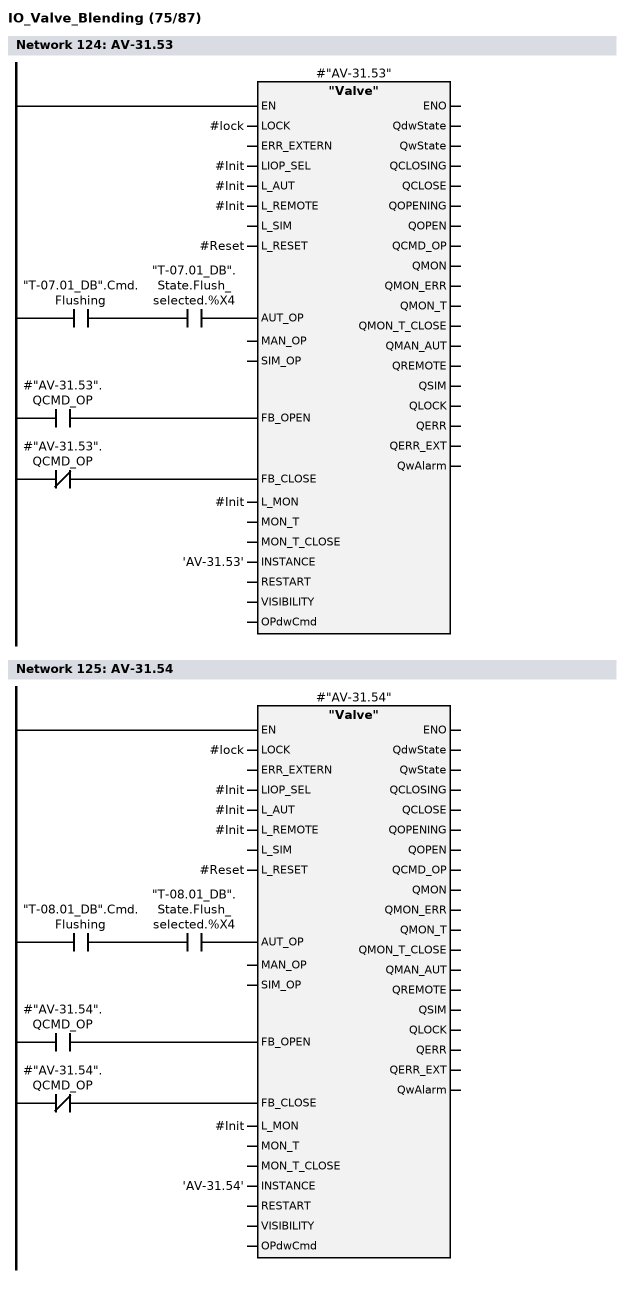
   RUNG wire#powerrail
      #"AV-31.53"(AUT_OP := wire#w1, FB_OPEN := wire#w2, FB_CLOSE := wire#w3, LOCK := #lock, ERR_EXTERN :=, LIOP_SEL := #Init, L_AUT := #Init, L_REMOTE := #Init, L_SIM :=, L_RESET := #Reset, MAN_OP :=, SIM_OP :=, L_MON := #Init, MON_T :=, MON_T_CLOSE :=, INSTANCE := 'AV-31.53', RESTART :=, VISIBILITY :=, OPdwCmd :=, QdwState =>, QwState =>, QCLOSING =>, QCLOSE =>, QOPENING =>, QOPEN =>, QCMD_OP =>, QMON =>, QMON_ERR =>, QMON_T =>, QMON_T_CLOSE =>, QMAN_AUT =>, QREMOTE =>, QSIM =>, QLOCK =>, QERR =>, QERR_EXT =>, QwAlarm =>)
   END_RUNG
   RUNG wire#powerrail
      Contact( "T-07.01_DB".Cmd.Flushing )
      Contact( "T-07.01_DB".State.Flush_selected.%X4 )
   END_RUNG wire#w1
   RUNG wire#powerrail
      Contact( #"AV-31.53".QCMD_OP )
   END_RUNG wire#w2
   RUNG wire#powerrail
      I_Contact( #"AV-31.53".QCMD_OP )
   END_RUNG wire#w3
   // the same network as SCL:
   #"AV-31.53"(LOCK := #lock,   // "Valve"
               LIOP_SEL := #Init,
               L_AUT := #Init,
               L_REMOTE := #Init,
               L_RESET := #Reset,
               AUT_OP := "T-07.01_DB".Cmd.Flushing AND "T-07.01_DB".State.Flush_selected.%X4,
               FB_OPEN := #"AV-31.53".QCMD_OP,
               FB_CLOSE := NOT #"AV-31.53".QCMD_OP,
               L_MON := #Init,
               INSTANCE := 'AV-31.53');
END_REGION

REGION Network 125: AV-31.54
   RUNG wire#powerrail
      #"AV-31.54"(AUT_OP := wire#w1, FB_OPEN := wire#w2, FB_CLOSE := wire#w3, LOCK := #lock, ERR_EXTERN :=, LIOP_SEL := #Init, L_AUT := #Init, L_REMOTE := #Init, L_SIM :=, L_RESET := #Reset, MAN_OP :=, SIM_OP :=, L_MON := #Init, MON_T :=, MON_T_CLOSE :=, INSTANCE := 'AV-31.54', RESTART :=, VISIBILITY :=, OPdwCmd :=, QdwState =>, QwState =>, QCLOSING =>, QCLOSE =>, QOPENING =>, QOPEN =>, QCMD_OP =>, QMON =>, QMON_ERR =>, QMON_T =>, QMON_T_CLOSE =>, QMAN_AUT =>, QREMOTE =>, QSIM =>, QLOCK =>, QERR =>, QERR_EXT =>, QwAlarm =>)
   END_RUNG
   RUNG wire#powerrail
      Contact( "T-08.01_DB".Cmd.Flushing )
      Contact( "T-08.01_DB".State.Flush_selected.%X4 )
   END_RUNG wire#w1
   RUNG wire#powerrail
      Contact( #"AV-31.54".QCMD_OP )
   END_RUNG wire#w2
   RUNG wire#powerrail
      I_Contact( #"AV-31.54".QCMD_OP )
   END_RUNG wire#w3
   // the same network as SCL:
   #"AV-31.54"(LOCK := #lock,   // "Valve"
               LIOP_SEL := #Init,
               L_AUT := #Init,
               L_REMOTE := #Init,
               L_RESET := #Reset,
               AUT_OP := "T-08.01_DB".Cmd.Flushing AND "T-08.01_DB".State.Flush_selected.%X4,
               FB_OPEN := #"AV-31.54".QCMD_OP,
               FB_CLOSE := NOT #"AV-31.54".QCMD_OP,
               L_MON := #Init,
               INSTANCE := 'AV-31.54');
END_REGION

REGION Network 126: AV-31.55
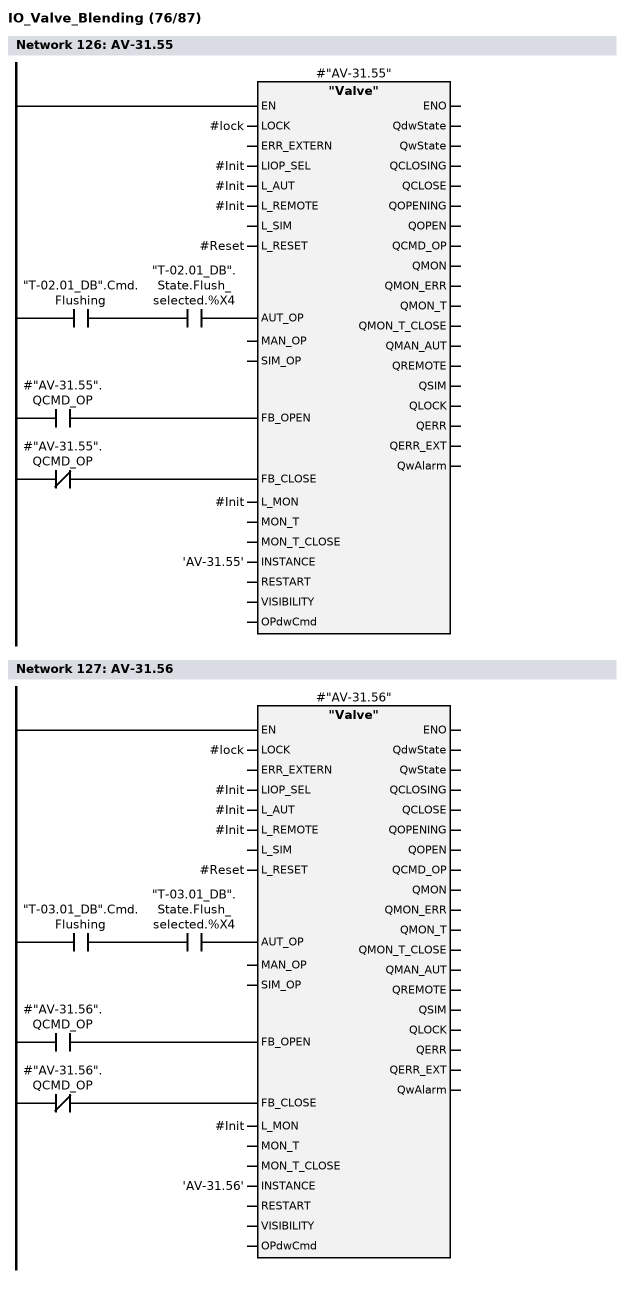
   RUNG wire#powerrail
      #"AV-31.55"(AUT_OP := wire#w1, FB_OPEN := wire#w2, FB_CLOSE := wire#w3, LOCK := #lock, ERR_EXTERN :=, LIOP_SEL := #Init, L_AUT := #Init, L_REMOTE := #Init, L_SIM :=, L_RESET := #Reset, MAN_OP :=, SIM_OP :=, L_MON := #Init, MON_T :=, MON_T_CLOSE :=, INSTANCE := 'AV-31.55', RESTART :=, VISIBILITY :=, OPdwCmd :=, QdwState =>, QwState =>, QCLOSING =>, QCLOSE =>, QOPENING =>, QOPEN =>, QCMD_OP =>, QMON =>, QMON_ERR =>, QMON_T =>, QMON_T_CLOSE =>, QMAN_AUT =>, QREMOTE =>, QSIM =>, QLOCK =>, QERR =>, QERR_EXT =>, QwAlarm =>)
   END_RUNG
   RUNG wire#powerrail
      Contact( "T-02.01_DB".Cmd.Flushing )
      Contact( "T-02.01_DB".State.Flush_selected.%X4 )
   END_RUNG wire#w1
   RUNG wire#powerrail
      Contact( #"AV-31.55".QCMD_OP )
   END_RUNG wire#w2
   RUNG wire#powerrail
      I_Contact( #"AV-31.55".QCMD_OP )
   END_RUNG wire#w3
   // the same network as SCL:
   #"AV-31.55"(LOCK := #lock,   // "Valve"
               LIOP_SEL := #Init,
               L_AUT := #Init,
               L_REMOTE := #Init,
               L_RESET := #Reset,
               AUT_OP := "T-02.01_DB".Cmd.Flushing AND "T-02.01_DB".State.Flush_selected.%X4,
               FB_OPEN := #"AV-31.55".QCMD_OP,
               FB_CLOSE := NOT #"AV-31.55".QCMD_OP,
               L_MON := #Init,
               INSTANCE := 'AV-31.55');
END_REGION

REGION Network 127: AV-31.56
   RUNG wire#powerrail
      #"AV-31.56"(AUT_OP := wire#w1, FB_OPEN := wire#w2, FB_CLOSE := wire#w3, LOCK := #lock, ERR_EXTERN :=, LIOP_SEL := #Init, L_AUT := #Init, L_REMOTE := #Init, L_SIM :=, L_RESET := #Reset, MAN_OP :=, SIM_OP :=, L_MON := #Init, MON_T :=, MON_T_CLOSE :=, INSTANCE := 'AV-31.56', RESTART :=, VISIBILITY :=, OPdwCmd :=, QdwState =>, QwState =>, QCLOSING =>, QCLOSE =>, QOPENING =>, QOPEN =>, QCMD_OP =>, QMON =>, QMON_ERR =>, QMON_T =>, QMON_T_CLOSE =>, QMAN_AUT =>, QREMOTE =>, QSIM =>, QLOCK =>, QERR =>, QERR_EXT =>, QwAlarm =>)
   END_RUNG
   RUNG wire#powerrail
      Contact( "T-03.01_DB".Cmd.Flushing )
      Contact( "T-03.01_DB".State.Flush_selected.%X4 )
   END_RUNG wire#w1
   RUNG wire#powerrail
      Contact( #"AV-31.56".QCMD_OP )
   END_RUNG wire#w2
   RUNG wire#powerrail
      I_Contact( #"AV-31.56".QCMD_OP )
   END_RUNG wire#w3
   // the same network as SCL:
   #"AV-31.56"(LOCK := #lock,   // "Valve"
               LIOP_SEL := #Init,
               L_AUT := #Init,
               L_REMOTE := #Init,
               L_RESET := #Reset,
               AUT_OP := "T-03.01_DB".Cmd.Flushing AND "T-03.01_DB".State.Flush_selected.%X4,
               FB_OPEN := #"AV-31.56".QCMD_OP,
               FB_CLOSE := NOT #"AV-31.56".QCMD_OP,
               L_MON := #Init,
               INSTANCE := 'AV-31.56');
END_REGION

REGION Network 128: AV-31.57
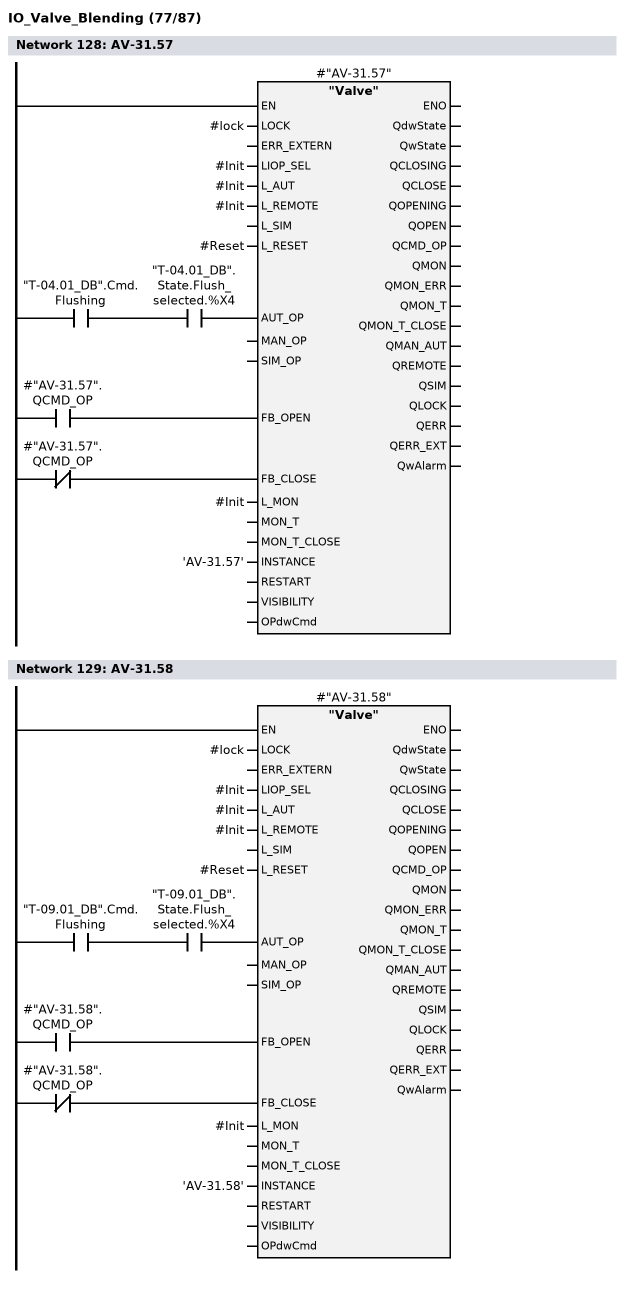
   RUNG wire#powerrail
      #"AV-31.57"(AUT_OP := wire#w1, FB_OPEN := wire#w2, FB_CLOSE := wire#w3, LOCK := #lock, ERR_EXTERN :=, LIOP_SEL := #Init, L_AUT := #Init, L_REMOTE := #Init, L_SIM :=, L_RESET := #Reset, MAN_OP :=, SIM_OP :=, L_MON := #Init, MON_T :=, MON_T_CLOSE :=, INSTANCE := 'AV-31.57', RESTART :=, VISIBILITY :=, OPdwCmd :=, QdwState =>, QwState =>, QCLOSING =>, QCLOSE =>, QOPENING =>, QOPEN =>, QCMD_OP =>, QMON =>, QMON_ERR =>, QMON_T =>, QMON_T_CLOSE =>, QMAN_AUT =>, QREMOTE =>, QSIM =>, QLOCK =>, QERR =>, QERR_EXT =>, QwAlarm =>)
   END_RUNG
   RUNG wire#powerrail
      Contact( "T-04.01_DB".Cmd.Flushing )
      Contact( "T-04.01_DB".State.Flush_selected.%X4 )
   END_RUNG wire#w1
   RUNG wire#powerrail
      Contact( #"AV-31.57".QCMD_OP )
   END_RUNG wire#w2
   RUNG wire#powerrail
      I_Contact( #"AV-31.57".QCMD_OP )
   END_RUNG wire#w3
   // the same network as SCL:
   #"AV-31.57"(LOCK := #lock,   // "Valve"
               LIOP_SEL := #Init,
               L_AUT := #Init,
               L_REMOTE := #Init,
               L_RESET := #Reset,
               AUT_OP := "T-04.01_DB".Cmd.Flushing AND "T-04.01_DB".State.Flush_selected.%X4,
               FB_OPEN := #"AV-31.57".QCMD_OP,
               FB_CLOSE := NOT #"AV-31.57".QCMD_OP,
               L_MON := #Init,
               INSTANCE := 'AV-31.57');
END_REGION

REGION Network 129: AV-31.58
   RUNG wire#powerrail
      #"AV-31.58"(AUT_OP := wire#w1, FB_OPEN := wire#w2, FB_CLOSE := wire#w3, LOCK := #lock, ERR_EXTERN :=, LIOP_SEL := #Init, L_AUT := #Init, L_REMOTE := #Init, L_SIM :=, L_RESET := #Reset, MAN_OP :=, SIM_OP :=, L_MON := #Init, MON_T :=, MON_T_CLOSE :=, INSTANCE := 'AV-31.58', RESTART :=, VISIBILITY :=, OPdwCmd :=, QdwState =>, QwState =>, QCLOSING =>, QCLOSE =>, QOPENING =>, QOPEN =>, QCMD_OP =>, QMON =>, QMON_ERR =>, QMON_T =>, QMON_T_CLOSE =>, QMAN_AUT =>, QREMOTE =>, QSIM =>, QLOCK =>, QERR =>, QERR_EXT =>, QwAlarm =>)
   END_RUNG
   RUNG wire#powerrail
      Contact( "T-09.01_DB".Cmd.Flushing )
      Contact( "T-09.01_DB".State.Flush_selected.%X4 )
   END_RUNG wire#w1
   RUNG wire#powerrail
      Contact( #"AV-31.58".QCMD_OP )
   END_RUNG wire#w2
   RUNG wire#powerrail
      I_Contact( #"AV-31.58".QCMD_OP )
   END_RUNG wire#w3
   // the same network as SCL:
   #"AV-31.58"(LOCK := #lock,   // "Valve"
               LIOP_SEL := #Init,
               L_AUT := #Init,
               L_REMOTE := #Init,
               L_RESET := #Reset,
               AUT_OP := "T-09.01_DB".Cmd.Flushing AND "T-09.01_DB".State.Flush_selected.%X4,
               FB_OPEN := #"AV-31.58".QCMD_OP,
               FB_CLOSE := NOT #"AV-31.58".QCMD_OP,
               L_MON := #Init,
               INSTANCE := 'AV-31.58');
END_REGION

REGION Network 130: AV-31.59
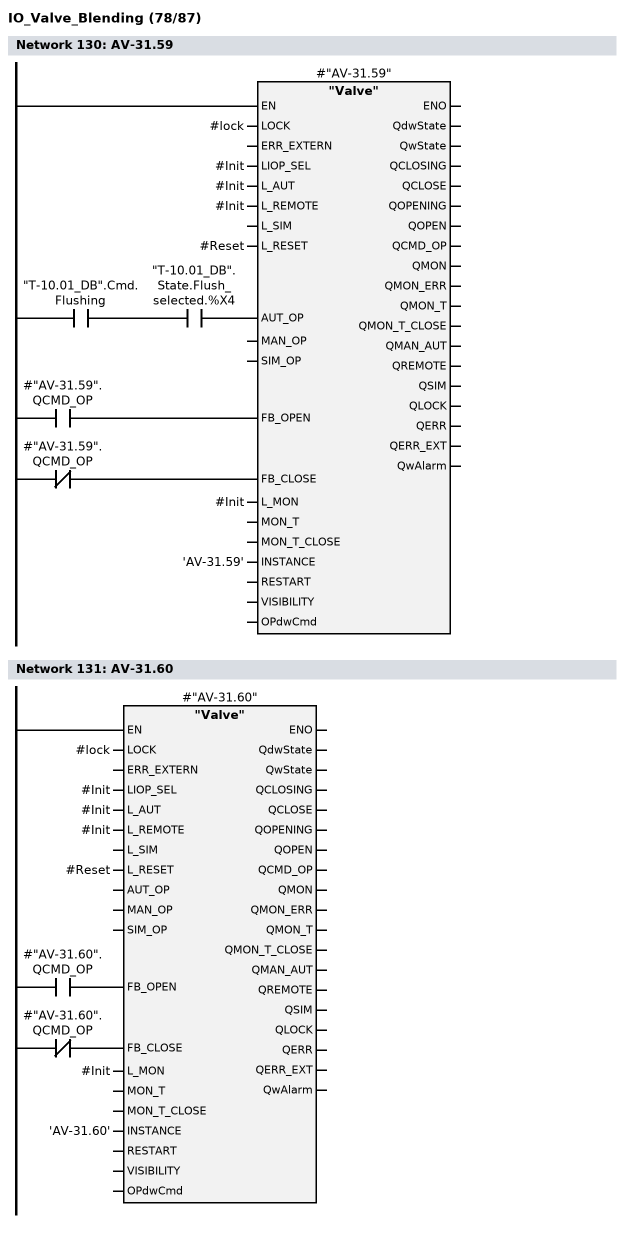
   RUNG wire#powerrail
      #"AV-31.59"(AUT_OP := wire#w1, FB_OPEN := wire#w2, FB_CLOSE := wire#w3, LOCK := #lock, ERR_EXTERN :=, LIOP_SEL := #Init, L_AUT := #Init, L_REMOTE := #Init, L_SIM :=, L_RESET := #Reset, MAN_OP :=, SIM_OP :=, L_MON := #Init, MON_T :=, MON_T_CLOSE :=, INSTANCE := 'AV-31.59', RESTART :=, VISIBILITY :=, OPdwCmd :=, QdwState =>, QwState =>, QCLOSING =>, QCLOSE =>, QOPENING =>, QOPEN =>, QCMD_OP =>, QMON =>, QMON_ERR =>, QMON_T =>, QMON_T_CLOSE =>, QMAN_AUT =>, QREMOTE =>, QSIM =>, QLOCK =>, QERR =>, QERR_EXT =>, QwAlarm =>)
   END_RUNG
   RUNG wire#powerrail
      Contact( "T-10.01_DB".Cmd.Flushing )
      Contact( "T-10.01_DB".State.Flush_selected.%X4 )
   END_RUNG wire#w1
   RUNG wire#powerrail
      Contact( #"AV-31.59".QCMD_OP )
   END_RUNG wire#w2
   RUNG wire#powerrail
      I_Contact( #"AV-31.59".QCMD_OP )
   END_RUNG wire#w3
   // the same network as SCL:
   #"AV-31.59"(LOCK := #lock,   // "Valve"
               LIOP_SEL := #Init,
               L_AUT := #Init,
               L_REMOTE := #Init,
               L_RESET := #Reset,
               AUT_OP := "T-10.01_DB".Cmd.Flushing AND "T-10.01_DB".State.Flush_selected.%X4,
               FB_OPEN := #"AV-31.59".QCMD_OP,
               FB_CLOSE := NOT #"AV-31.59".QCMD_OP,
               L_MON := #Init,
               INSTANCE := 'AV-31.59');
END_REGION

REGION Network 131: AV-31.60
   RUNG wire#powerrail
      #"AV-31.60"(FB_OPEN := wire#w1, FB_CLOSE := wire#w2, LOCK := #lock, ERR_EXTERN :=, LIOP_SEL := #Init, L_AUT := #Init, L_REMOTE := #Init, L_SIM :=, L_RESET := #Reset, AUT_OP :=, MAN_OP :=, SIM_OP :=, L_MON := #Init, MON_T :=, MON_T_CLOSE :=, INSTANCE := 'AV-31.60', RESTART :=, VISIBILITY :=, OPdwCmd :=, QdwState =>, QwState =>, QCLOSING =>, QCLOSE =>, QOPENING =>, QOPEN =>, QCMD_OP =>, QMON =>, QMON_ERR =>, QMON_T =>, QMON_T_CLOSE =>, QMAN_AUT =>, QREMOTE =>, QSIM =>, QLOCK =>, QERR =>, QERR_EXT =>, QwAlarm =>)
   END_RUNG
   RUNG wire#powerrail
      Contact( #"AV-31.60".QCMD_OP )
   END_RUNG wire#w1
   RUNG wire#powerrail
      I_Contact( #"AV-31.60".QCMD_OP )
   END_RUNG wire#w2
   // the same network as SCL:
   #"AV-31.60"(LOCK := #lock,   // "Valve"
               LIOP_SEL := #Init,
               L_AUT := #Init,
               L_REMOTE := #Init,
               L_RESET := #Reset,
               FB_OPEN := #"AV-31.60".QCMD_OP,
               FB_CLOSE := NOT #"AV-31.60".QCMD_OP,
               L_MON := #Init,
               INSTANCE := 'AV-31.60');
END_REGION

REGION Network 132: AV-31.61
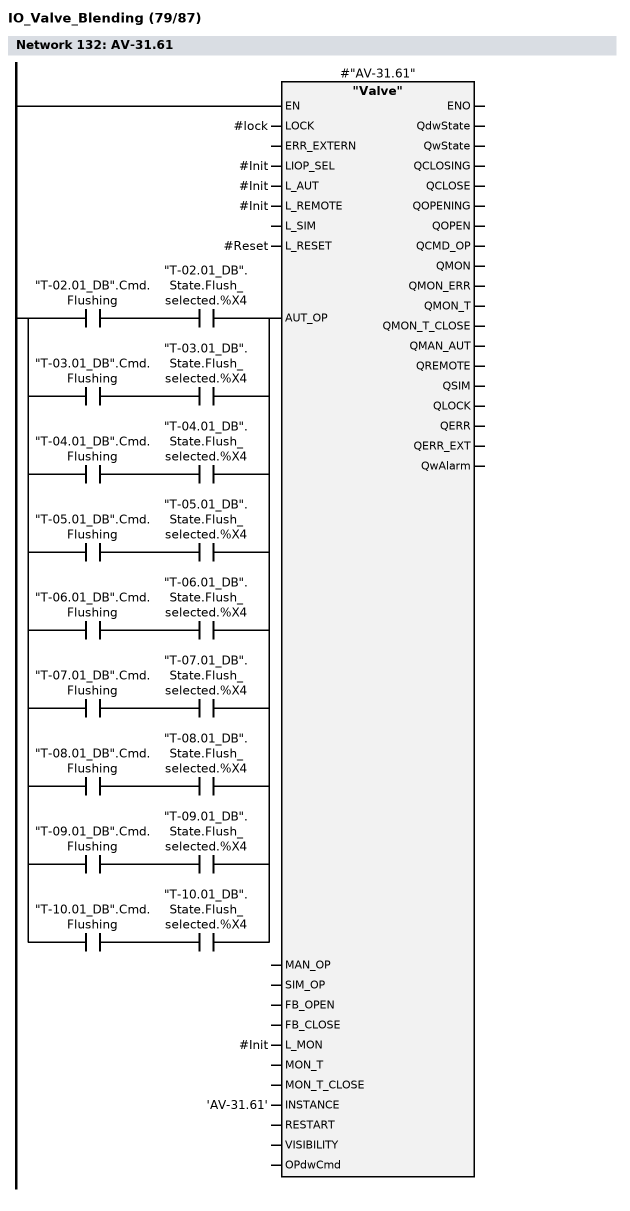
   RUNG wire#powerrail
      #"AV-31.61"(AUT_OP := wire#w1, LOCK := #lock, ERR_EXTERN :=, LIOP_SEL := #Init, L_AUT := #Init, L_REMOTE := #Init, L_SIM :=, L_RESET := #Reset, MAN_OP :=, SIM_OP :=, FB_OPEN :=, FB_CLOSE :=, L_MON := #Init, MON_T :=, MON_T_CLOSE :=, INSTANCE := 'AV-31.61', RESTART :=, VISIBILITY :=, OPdwCmd :=, QdwState =>, QwState =>, QCLOSING =>, QCLOSE =>, QOPENING =>, QOPEN =>, QCMD_OP =>, QMON =>, QMON_ERR =>, QMON_T =>, QMON_T_CLOSE =>, QMAN_AUT =>, QREMOTE =>, QSIM =>, QLOCK =>, QERR =>, QERR_EXT =>, QwAlarm =>)
   END_RUNG
   RUNG wire#powerrail
      Contact( "T-02.01_DB".Cmd.Flushing )
      Contact( "T-02.01_DB".State.Flush_selected.%X4 )
   END_RUNG wire#w1
   RUNG wire#powerrail
      Contact( "T-03.01_DB".Cmd.Flushing )
      Contact( "T-03.01_DB".State.Flush_selected.%X4 )
   END_RUNG wire#w1
   RUNG wire#powerrail
      Contact( "T-04.01_DB".Cmd.Flushing )
      Contact( "T-04.01_DB".State.Flush_selected.%X4 )
   END_RUNG wire#w1
   RUNG wire#powerrail
      Contact( "T-05.01_DB".Cmd.Flushing )
      Contact( "T-05.01_DB".State.Flush_selected.%X4 )
   END_RUNG wire#w1
   RUNG wire#powerrail
      Contact( "T-06.01_DB".Cmd.Flushing )
      Contact( "T-06.01_DB".State.Flush_selected.%X4 )
   END_RUNG wire#w1
   RUNG wire#powerrail
      Contact( "T-07.01_DB".Cmd.Flushing )
      Contact( "T-07.01_DB".State.Flush_selected.%X4 )
   END_RUNG wire#w1
   RUNG wire#powerrail
      Contact( "T-08.01_DB".Cmd.Flushing )
      Contact( "T-08.01_DB".State.Flush_selected.%X4 )
   END_RUNG wire#w1
   RUNG wire#powerrail
      Contact( "T-09.01_DB".Cmd.Flushing )
      Contact( "T-09.01_DB".State.Flush_selected.%X4 )
   END_RUNG wire#w1
   RUNG wire#powerrail
      Contact( "T-10.01_DB".Cmd.Flushing )
      Contact( "T-10.01_DB".State.Flush_selected.%X4 )
   END_RUNG wire#w1
   // the same network as SCL:
   #"AV-31.61"(LOCK := #lock,   // "Valve"
               LIOP_SEL := #Init,
               L_AUT := #Init,
               L_REMOTE := #Init,
               L_RESET := #Reset,
               AUT_OP := ("T-02.01_DB".Cmd.Flushing AND "T-02.01_DB".State.Flush_selected.%X4) OR ("T-03.01_DB".Cmd.Flushing AND "T-03.01_DB".State.Flush_selected.%X4) OR ("T-04.01_DB".Cmd.Flushing AND "T-04.01_DB".State.Flush_selected.%X4) OR ("T-05.01_DB".Cmd.Flushing AND "T-05.01_DB".State.Flush_selected.%X4) OR ("T-06.01_DB".Cmd.Flushing AND "T-06.01_DB".State.Flush_selected.%X4) OR ("T-07.01_DB".Cmd.Flushing AND "T-07.01_DB".State.Flush_selected.%X4) OR ("T-08.01_DB".Cmd.Flushing AND "T-08.01_DB".State.Flush_selected.%X4) OR ("T-09.01_DB".Cmd.Flushing AND "T-09.01_DB".State.Flush_selected.%X4) OR ("T-10.01_DB".Cmd.Flushing AND "T-10.01_DB".State.Flush_selected.%X4),
               L_MON := #Init,
               INSTANCE := 'AV-31.61');
END_REGION

REGION Network 133: AV-31.62
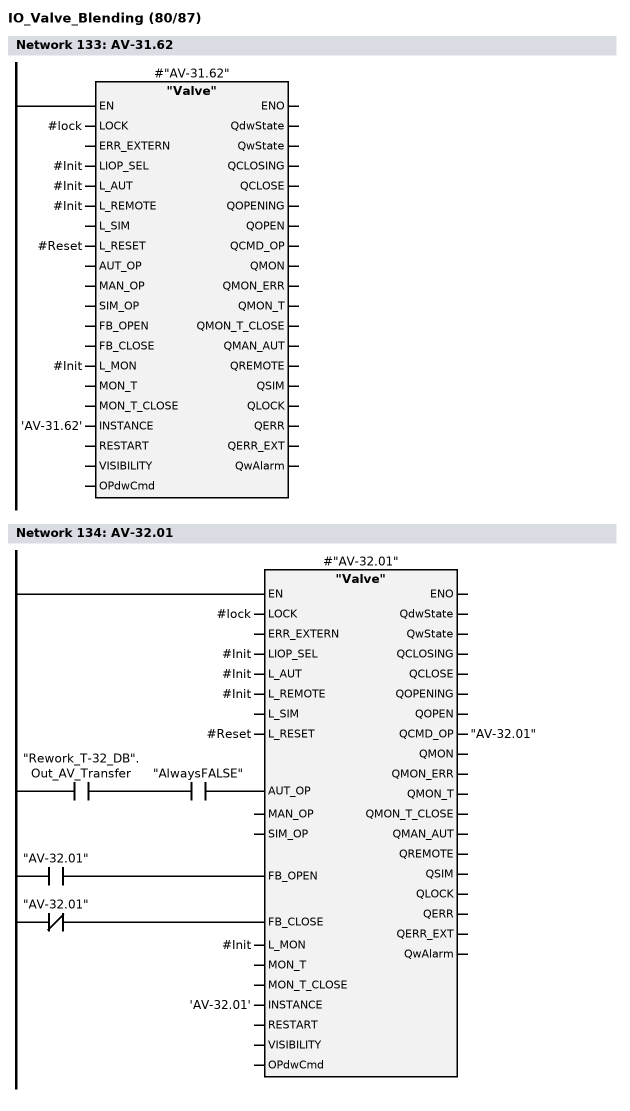
   RUNG wire#powerrail
      #"AV-31.62"(LOCK := #lock, ERR_EXTERN :=, LIOP_SEL := #Init, L_AUT := #Init, L_REMOTE := #Init, L_SIM :=, L_RESET := #Reset, AUT_OP :=, MAN_OP :=, SIM_OP :=, FB_OPEN :=, FB_CLOSE :=, L_MON := #Init, MON_T :=, MON_T_CLOSE :=, INSTANCE := 'AV-31.62', RESTART :=, VISIBILITY :=, OPdwCmd :=, QdwState =>, QwState =>, QCLOSING =>, QCLOSE =>, QOPENING =>, QOPEN =>, QCMD_OP =>, QMON =>, QMON_ERR =>, QMON_T =>, QMON_T_CLOSE =>, QMAN_AUT =>, QREMOTE =>, QSIM =>, QLOCK =>, QERR =>, QERR_EXT =>, QwAlarm =>)
   END_RUNG
   // the same network as SCL:
   #"AV-31.62"(LOCK := #lock,   // "Valve"
               LIOP_SEL := #Init,
               L_AUT := #Init,
               L_REMOTE := #Init,
               L_RESET := #Reset,
               L_MON := #Init,
               INSTANCE := 'AV-31.62');
END_REGION

REGION Network 134: AV-32.01
   RUNG wire#powerrail
      #"AV-32.01"(AUT_OP := wire#w1, FB_OPEN := wire#w2, FB_CLOSE := wire#w3, LOCK := #lock, ERR_EXTERN :=, LIOP_SEL := #Init, L_AUT := #Init, L_REMOTE := #Init, L_SIM :=, L_RESET := #Reset, MAN_OP :=, SIM_OP :=, L_MON := #Init, MON_T :=, MON_T_CLOSE :=, INSTANCE := 'AV-32.01', RESTART :=, VISIBILITY :=, OPdwCmd :=, QdwState =>, QwState =>, QCLOSING =>, QCLOSE =>, QOPENING =>, QOPEN =>, QCMD_OP => "AV-32.01", QMON =>, QMON_ERR =>, QMON_T =>, QMON_T_CLOSE =>, QMAN_AUT =>, QREMOTE =>, QSIM =>, QLOCK =>, QERR =>, QERR_EXT =>, QwAlarm =>)
   END_RUNG
   RUNG wire#powerrail
      Contact( "Rework_T-32_DB".Out_AV_Transfer )
      Contact( "AlwaysFALSE" )
   END_RUNG wire#w1
   RUNG wire#powerrail
      Contact( "AV-32.01" )
   END_RUNG wire#w2
   RUNG wire#powerrail
      I_Contact( "AV-32.01" )
   END_RUNG wire#w3
   // the same network as SCL:
   #"AV-32.01"(LOCK := #lock,   // "Valve"
               LIOP_SEL := #Init,
               L_AUT := #Init,
               L_REMOTE := #Init,
               L_RESET := #Reset,
               AUT_OP := "Rework_T-32_DB".Out_AV_Transfer AND "AlwaysFALSE",
               FB_OPEN := "AV-32.01",
               FB_CLOSE := NOT "AV-32.01",
               L_MON := #Init,
               INSTANCE := 'AV-32.01',
               QCMD_OP => "AV-32.01");
END_REGION

REGION Network 135: AV-32.02
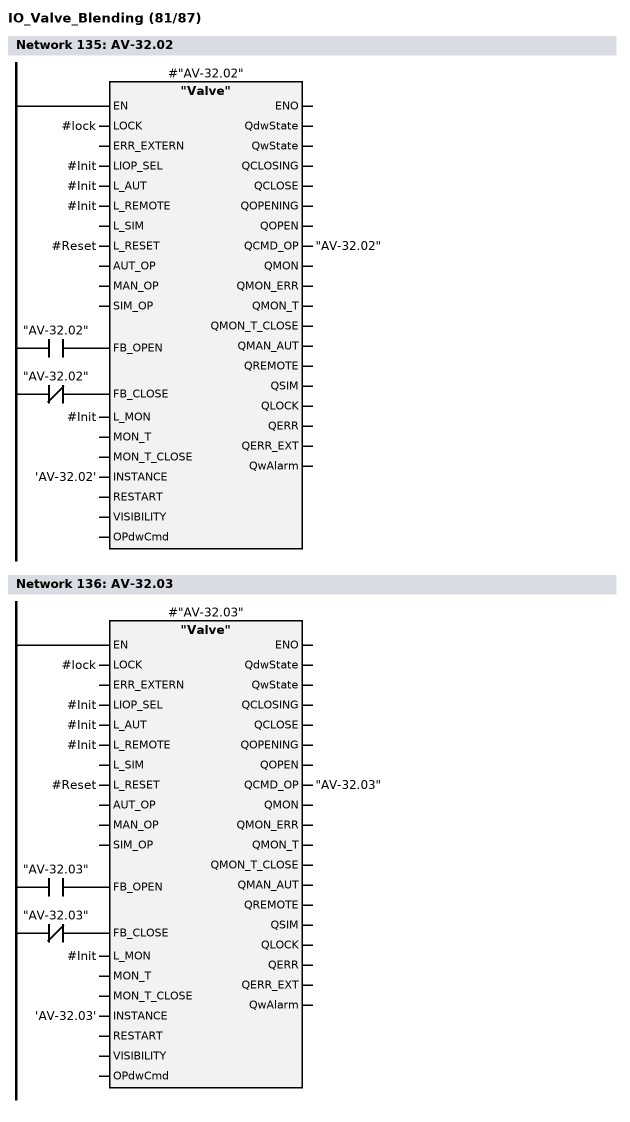
   RUNG wire#powerrail
      #"AV-32.02"(FB_OPEN := wire#w1, FB_CLOSE := wire#w2, LOCK := #lock, ERR_EXTERN :=, LIOP_SEL := #Init, L_AUT := #Init, L_REMOTE := #Init, L_SIM :=, L_RESET := #Reset, AUT_OP :=, MAN_OP :=, SIM_OP :=, L_MON := #Init, MON_T :=, MON_T_CLOSE :=, INSTANCE := 'AV-32.02', RESTART :=, VISIBILITY :=, OPdwCmd :=, QdwState =>, QwState =>, QCLOSING =>, QCLOSE =>, QOPENING =>, QOPEN =>, QCMD_OP => "AV-32.02", QMON =>, QMON_ERR =>, QMON_T =>, QMON_T_CLOSE =>, QMAN_AUT =>, QREMOTE =>, QSIM =>, QLOCK =>, QERR =>, QERR_EXT =>, QwAlarm =>)
   END_RUNG
   RUNG wire#powerrail
      Contact( "AV-32.02" )
   END_RUNG wire#w1
   RUNG wire#powerrail
      I_Contact( "AV-32.02" )
   END_RUNG wire#w2
   // the same network as SCL:
   #"AV-32.02"(LOCK := #lock,   // "Valve"
               LIOP_SEL := #Init,
               L_AUT := #Init,
               L_REMOTE := #Init,
               L_RESET := #Reset,
               FB_OPEN := "AV-32.02",
               FB_CLOSE := NOT "AV-32.02",
               L_MON := #Init,
               INSTANCE := 'AV-32.02',
               QCMD_OP => "AV-32.02");
END_REGION

REGION Network 136: AV-32.03
   RUNG wire#powerrail
      #"AV-32.03"(FB_OPEN := wire#w1, FB_CLOSE := wire#w2, LOCK := #lock, ERR_EXTERN :=, LIOP_SEL := #Init, L_AUT := #Init, L_REMOTE := #Init, L_SIM :=, L_RESET := #Reset, AUT_OP :=, MAN_OP :=, SIM_OP :=, L_MON := #Init, MON_T :=, MON_T_CLOSE :=, INSTANCE := 'AV-32.03', RESTART :=, VISIBILITY :=, OPdwCmd :=, QdwState =>, QwState =>, QCLOSING =>, QCLOSE =>, QOPENING =>, QOPEN =>, QCMD_OP => "AV-32.03", QMON =>, QMON_ERR =>, QMON_T =>, QMON_T_CLOSE =>, QMAN_AUT =>, QREMOTE =>, QSIM =>, QLOCK =>, QERR =>, QERR_EXT =>, QwAlarm =>)
   END_RUNG
   RUNG wire#powerrail
      Contact( "AV-32.03" )
   END_RUNG wire#w1
   RUNG wire#powerrail
      I_Contact( "AV-32.03" )
   END_RUNG wire#w2
   // the same network as SCL:
   #"AV-32.03"(LOCK := #lock,   // "Valve"
               LIOP_SEL := #Init,
               L_AUT := #Init,
               L_REMOTE := #Init,
               L_RESET := #Reset,
               FB_OPEN := "AV-32.03",
               FB_CLOSE := NOT "AV-32.03",
               L_MON := #Init,
               INSTANCE := 'AV-32.03',
               QCMD_OP => "AV-32.03");
END_REGION

REGION Network 137: AV-32.06
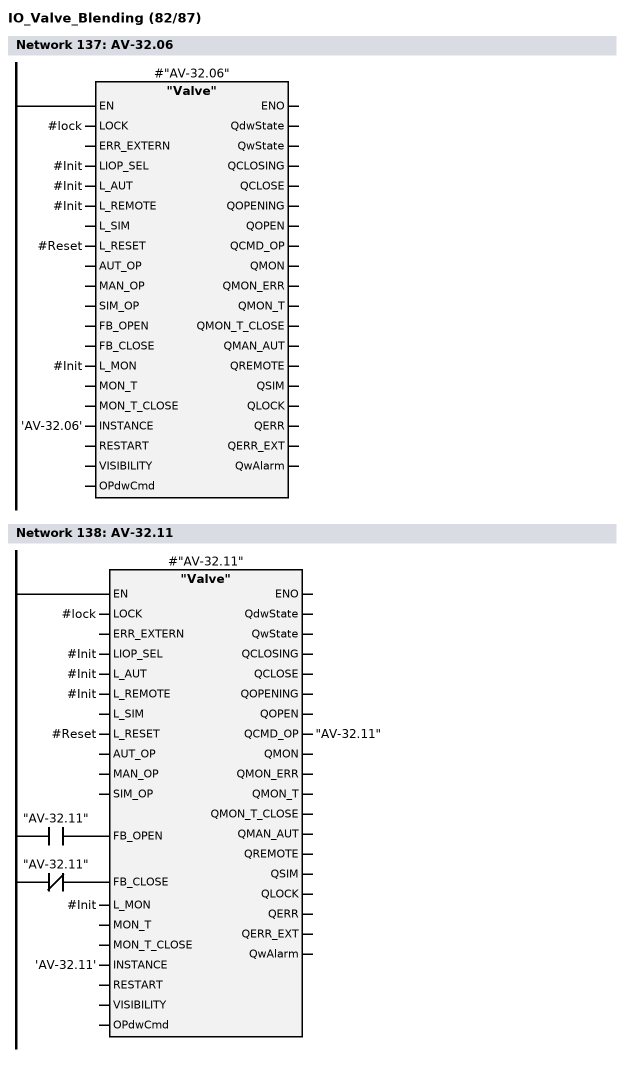
   RUNG wire#powerrail
      #"AV-32.06"(LOCK := #lock, ERR_EXTERN :=, LIOP_SEL := #Init, L_AUT := #Init, L_REMOTE := #Init, L_SIM :=, L_RESET := #Reset, AUT_OP :=, MAN_OP :=, SIM_OP :=, FB_OPEN :=, FB_CLOSE :=, L_MON := #Init, MON_T :=, MON_T_CLOSE :=, INSTANCE := 'AV-32.06', RESTART :=, VISIBILITY :=, OPdwCmd :=, QdwState =>, QwState =>, QCLOSING =>, QCLOSE =>, QOPENING =>, QOPEN =>, QCMD_OP =>, QMON =>, QMON_ERR =>, QMON_T =>, QMON_T_CLOSE =>, QMAN_AUT =>, QREMOTE =>, QSIM =>, QLOCK =>, QERR =>, QERR_EXT =>, QwAlarm =>)
   END_RUNG
   // the same network as SCL:
   #"AV-32.06"(LOCK := #lock,   // "Valve"
               LIOP_SEL := #Init,
               L_AUT := #Init,
               L_REMOTE := #Init,
               L_RESET := #Reset,
               L_MON := #Init,
               INSTANCE := 'AV-32.06');
END_REGION

REGION Network 138: AV-32.11
   RUNG wire#powerrail
      #"AV-32.11"(FB_OPEN := wire#w1, FB_CLOSE := wire#w2, LOCK := #lock, ERR_EXTERN :=, LIOP_SEL := #Init, L_AUT := #Init, L_REMOTE := #Init, L_SIM :=, L_RESET := #Reset, AUT_OP :=, MAN_OP :=, SIM_OP :=, L_MON := #Init, MON_T :=, MON_T_CLOSE :=, INSTANCE := 'AV-32.11', RESTART :=, VISIBILITY :=, OPdwCmd :=, QdwState =>, QwState =>, QCLOSING =>, QCLOSE =>, QOPENING =>, QOPEN =>, QCMD_OP => "AV-32.11", QMON =>, QMON_ERR =>, QMON_T =>, QMON_T_CLOSE =>, QMAN_AUT =>, QREMOTE =>, QSIM =>, QLOCK =>, QERR =>, QERR_EXT =>, QwAlarm =>)
   END_RUNG
   RUNG wire#powerrail
      Contact( "AV-32.11" )
   END_RUNG wire#w1
   RUNG wire#powerrail
      I_Contact( "AV-32.11" )
   END_RUNG wire#w2
   // the same network as SCL:
   #"AV-32.11"(LOCK := #lock,   // "Valve"
               LIOP_SEL := #Init,
               L_AUT := #Init,
               L_REMOTE := #Init,
               L_RESET := #Reset,
               FB_OPEN := "AV-32.11",
               FB_CLOSE := NOT "AV-32.11",
               L_MON := #Init,
               INSTANCE := 'AV-32.11',
               QCMD_OP => "AV-32.11");
END_REGION

REGION Network 139: AV-32.21
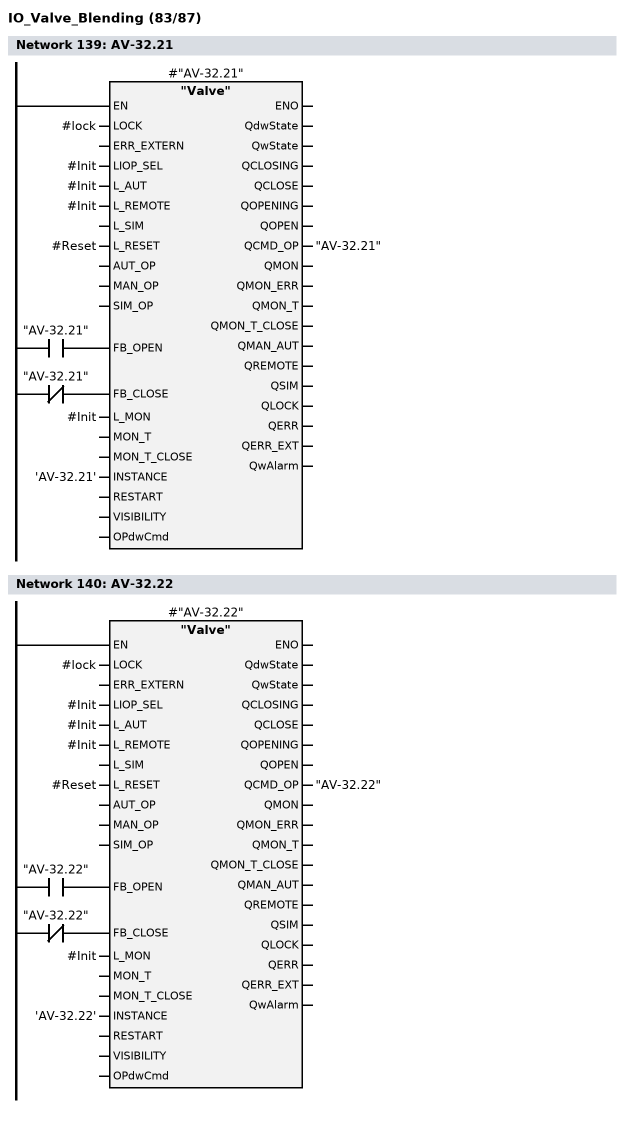
   RUNG wire#powerrail
      #"AV-32.21"(FB_OPEN := wire#w1, FB_CLOSE := wire#w2, LOCK := #lock, ERR_EXTERN :=, LIOP_SEL := #Init, L_AUT := #Init, L_REMOTE := #Init, L_SIM :=, L_RESET := #Reset, AUT_OP :=, MAN_OP :=, SIM_OP :=, L_MON := #Init, MON_T :=, MON_T_CLOSE :=, INSTANCE := 'AV-32.21', RESTART :=, VISIBILITY :=, OPdwCmd :=, QdwState =>, QwState =>, QCLOSING =>, QCLOSE =>, QOPENING =>, QOPEN =>, QCMD_OP => "AV-32.21", QMON =>, QMON_ERR =>, QMON_T =>, QMON_T_CLOSE =>, QMAN_AUT =>, QREMOTE =>, QSIM =>, QLOCK =>, QERR =>, QERR_EXT =>, QwAlarm =>)
   END_RUNG
   RUNG wire#powerrail
      Contact( "AV-32.21" )
   END_RUNG wire#w1
   RUNG wire#powerrail
      I_Contact( "AV-32.21" )
   END_RUNG wire#w2
   // the same network as SCL:
   #"AV-32.21"(LOCK := #lock,   // "Valve"
               LIOP_SEL := #Init,
               L_AUT := #Init,
               L_REMOTE := #Init,
               L_RESET := #Reset,
               FB_OPEN := "AV-32.21",
               FB_CLOSE := NOT "AV-32.21",
               L_MON := #Init,
               INSTANCE := 'AV-32.21',
               QCMD_OP => "AV-32.21");
END_REGION

REGION Network 140: AV-32.22
   RUNG wire#powerrail
      #"AV-32.22"(FB_OPEN := wire#w1, FB_CLOSE := wire#w2, LOCK := #lock, ERR_EXTERN :=, LIOP_SEL := #Init, L_AUT := #Init, L_REMOTE := #Init, L_SIM :=, L_RESET := #Reset, AUT_OP :=, MAN_OP :=, SIM_OP :=, L_MON := #Init, MON_T :=, MON_T_CLOSE :=, INSTANCE := 'AV-32.22', RESTART :=, VISIBILITY :=, OPdwCmd :=, QdwState =>, QwState =>, QCLOSING =>, QCLOSE =>, QOPENING =>, QOPEN =>, QCMD_OP => "AV-32.22", QMON =>, QMON_ERR =>, QMON_T =>, QMON_T_CLOSE =>, QMAN_AUT =>, QREMOTE =>, QSIM =>, QLOCK =>, QERR =>, QERR_EXT =>, QwAlarm =>)
   END_RUNG
   RUNG wire#powerrail
      Contact( "AV-32.22" )
   END_RUNG wire#w1
   RUNG wire#powerrail
      I_Contact( "AV-32.22" )
   END_RUNG wire#w2
   // the same network as SCL:
   #"AV-32.22"(LOCK := #lock,   // "Valve"
               LIOP_SEL := #Init,
               L_AUT := #Init,
               L_REMOTE := #Init,
               L_RESET := #Reset,
               FB_OPEN := "AV-32.22",
               FB_CLOSE := NOT "AV-32.22",
               L_MON := #Init,
               INSTANCE := 'AV-32.22',
               QCMD_OP => "AV-32.22");
END_REGION

REGION Network 141: AV-20.42
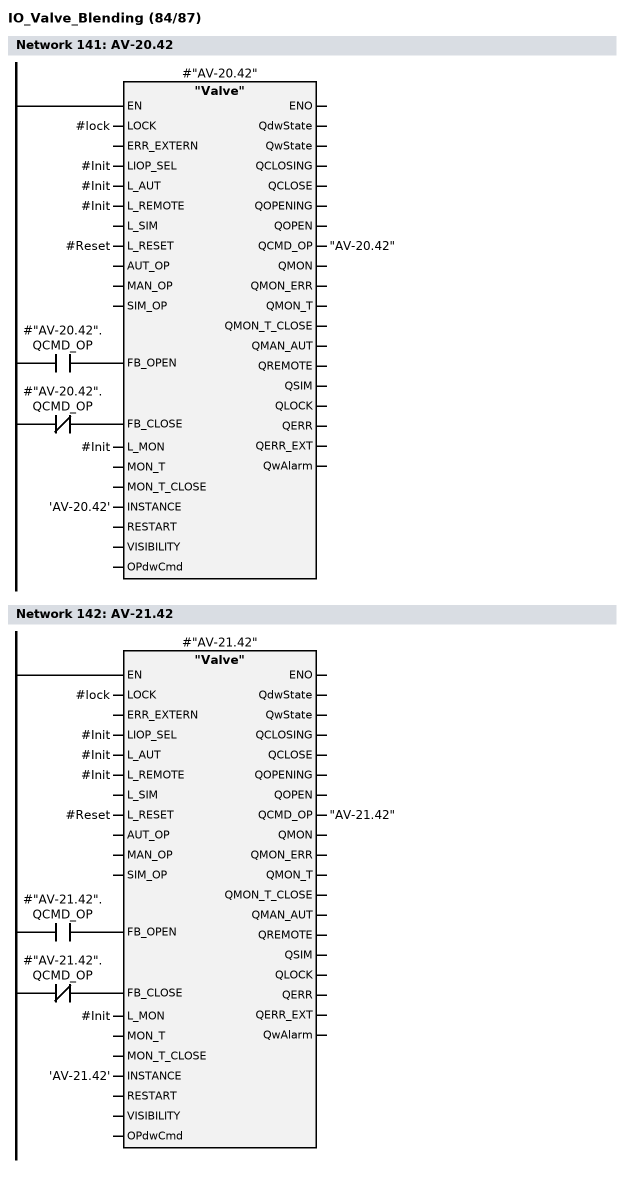
   RUNG wire#powerrail
      #"AV-20.42"(FB_OPEN := wire#w1, FB_CLOSE := wire#w2, LOCK := #lock, ERR_EXTERN :=, LIOP_SEL := #Init, L_AUT := #Init, L_REMOTE := #Init, L_SIM :=, L_RESET := #Reset, AUT_OP :=, MAN_OP :=, SIM_OP :=, L_MON := #Init, MON_T :=, MON_T_CLOSE :=, INSTANCE := 'AV-20.42', RESTART :=, VISIBILITY :=, OPdwCmd :=, QdwState =>, QwState =>, QCLOSING =>, QCLOSE =>, QOPENING =>, QOPEN =>, QCMD_OP => "AV-20.42", QMON =>, QMON_ERR =>, QMON_T =>, QMON_T_CLOSE =>, QMAN_AUT =>, QREMOTE =>, QSIM =>, QLOCK =>, QERR =>, QERR_EXT =>, QwAlarm =>)
   END_RUNG
   RUNG wire#powerrail
      Contact( #"AV-20.42".QCMD_OP )
   END_RUNG wire#w1
   RUNG wire#powerrail
      I_Contact( #"AV-20.42".QCMD_OP )
   END_RUNG wire#w2
   // the same network as SCL:
   #"AV-20.42"(LOCK := #lock,   // "Valve"
               LIOP_SEL := #Init,
               L_AUT := #Init,
               L_REMOTE := #Init,
               L_RESET := #Reset,
               FB_OPEN := #"AV-20.42".QCMD_OP,
               FB_CLOSE := NOT #"AV-20.42".QCMD_OP,
               L_MON := #Init,
               INSTANCE := 'AV-20.42',
               QCMD_OP => "AV-20.42");
END_REGION

REGION Network 142: AV-21.42
   RUNG wire#powerrail
      #"AV-21.42"(FB_OPEN := wire#w1, FB_CLOSE := wire#w2, LOCK := #lock, ERR_EXTERN :=, LIOP_SEL := #Init, L_AUT := #Init, L_REMOTE := #Init, L_SIM :=, L_RESET := #Reset, AUT_OP :=, MAN_OP :=, SIM_OP :=, L_MON := #Init, MON_T :=, MON_T_CLOSE :=, INSTANCE := 'AV-21.42', RESTART :=, VISIBILITY :=, OPdwCmd :=, QdwState =>, QwState =>, QCLOSING =>, QCLOSE =>, QOPENING =>, QOPEN =>, QCMD_OP => "AV-21.42", QMON =>, QMON_ERR =>, QMON_T =>, QMON_T_CLOSE =>, QMAN_AUT =>, QREMOTE =>, QSIM =>, QLOCK =>, QERR =>, QERR_EXT =>, QwAlarm =>)
   END_RUNG
   RUNG wire#powerrail
      Contact( #"AV-21.42".QCMD_OP )
   END_RUNG wire#w1
   RUNG wire#powerrail
      I_Contact( #"AV-21.42".QCMD_OP )
   END_RUNG wire#w2
   // the same network as SCL:
   #"AV-21.42"(LOCK := #lock,   // "Valve"
               LIOP_SEL := #Init,
               L_AUT := #Init,
               L_REMOTE := #Init,
               L_RESET := #Reset,
               FB_OPEN := #"AV-21.42".QCMD_OP,
               FB_CLOSE := NOT #"AV-21.42".QCMD_OP,
               L_MON := #Init,
               INSTANCE := 'AV-21.42',
               QCMD_OP => "AV-21.42");
END_REGION

REGION Network 143: AV-22.04
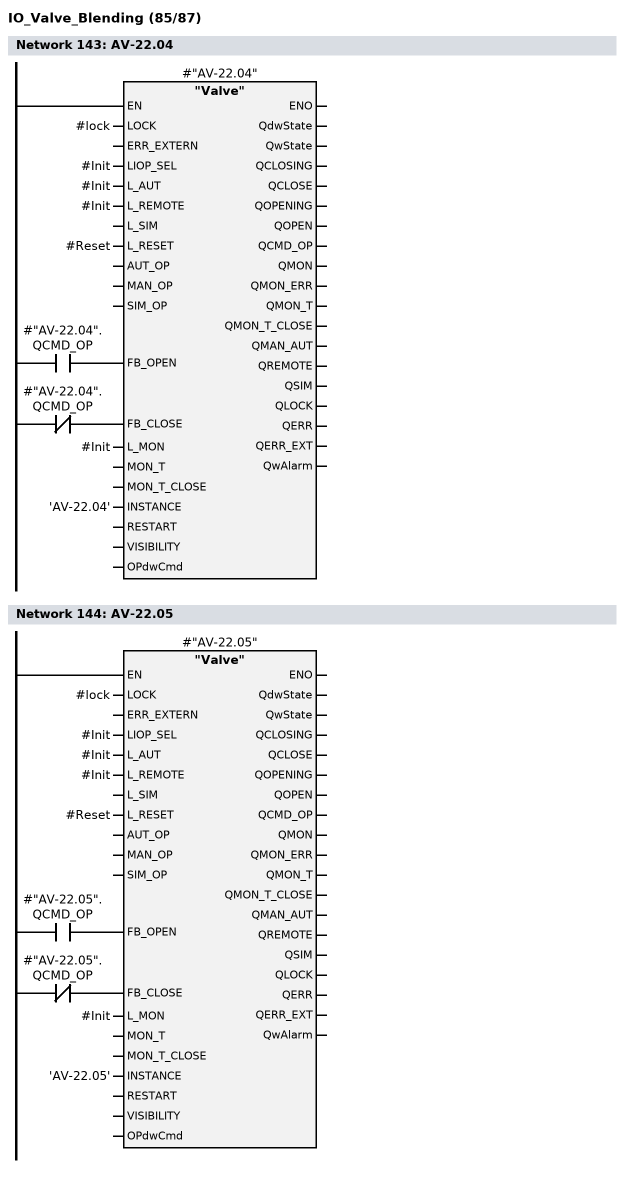
   RUNG wire#powerrail
      #"AV-22.04"(FB_OPEN := wire#w1, FB_CLOSE := wire#w2, LOCK := #lock, ERR_EXTERN :=, LIOP_SEL := #Init, L_AUT := #Init, L_REMOTE := #Init, L_SIM :=, L_RESET := #Reset, AUT_OP :=, MAN_OP :=, SIM_OP :=, L_MON := #Init, MON_T :=, MON_T_CLOSE :=, INSTANCE := 'AV-22.04', RESTART :=, VISIBILITY :=, OPdwCmd :=, QdwState =>, QwState =>, QCLOSING =>, QCLOSE =>, QOPENING =>, QOPEN =>, QCMD_OP =>, QMON =>, QMON_ERR =>, QMON_T =>, QMON_T_CLOSE =>, QMAN_AUT =>, QREMOTE =>, QSIM =>, QLOCK =>, QERR =>, QERR_EXT =>, QwAlarm =>)
   END_RUNG
   RUNG wire#powerrail
      Contact( #"AV-22.04".QCMD_OP )
   END_RUNG wire#w1
   RUNG wire#powerrail
      I_Contact( #"AV-22.04".QCMD_OP )
   END_RUNG wire#w2
   // the same network as SCL:
   #"AV-22.04"(LOCK := #lock,   // "Valve"
               LIOP_SEL := #Init,
               L_AUT := #Init,
               L_REMOTE := #Init,
               L_RESET := #Reset,
               FB_OPEN := #"AV-22.04".QCMD_OP,
               FB_CLOSE := NOT #"AV-22.04".QCMD_OP,
               L_MON := #Init,
               INSTANCE := 'AV-22.04');
END_REGION

REGION Network 144: AV-22.05
   RUNG wire#powerrail
      #"AV-22.05"(FB_OPEN := wire#w1, FB_CLOSE := wire#w2, LOCK := #lock, ERR_EXTERN :=, LIOP_SEL := #Init, L_AUT := #Init, L_REMOTE := #Init, L_SIM :=, L_RESET := #Reset, AUT_OP :=, MAN_OP :=, SIM_OP :=, L_MON := #Init, MON_T :=, MON_T_CLOSE :=, INSTANCE := 'AV-22.05', RESTART :=, VISIBILITY :=, OPdwCmd :=, QdwState =>, QwState =>, QCLOSING =>, QCLOSE =>, QOPENING =>, QOPEN =>, QCMD_OP =>, QMON =>, QMON_ERR =>, QMON_T =>, QMON_T_CLOSE =>, QMAN_AUT =>, QREMOTE =>, QSIM =>, QLOCK =>, QERR =>, QERR_EXT =>, QwAlarm =>)
   END_RUNG
   RUNG wire#powerrail
      Contact( #"AV-22.05".QCMD_OP )
   END_RUNG wire#w1
   RUNG wire#powerrail
      I_Contact( #"AV-22.05".QCMD_OP )
   END_RUNG wire#w2
   // the same network as SCL:
   #"AV-22.05"(LOCK := #lock,   // "Valve"
               LIOP_SEL := #Init,
               L_AUT := #Init,
               L_REMOTE := #Init,
               L_RESET := #Reset,
               FB_OPEN := #"AV-22.05".QCMD_OP,
               FB_CLOSE := NOT #"AV-22.05".QCMD_OP,
               L_MON := #Init,
               INSTANCE := 'AV-22.05');
END_REGION

REGION Network 145: AV-30.42
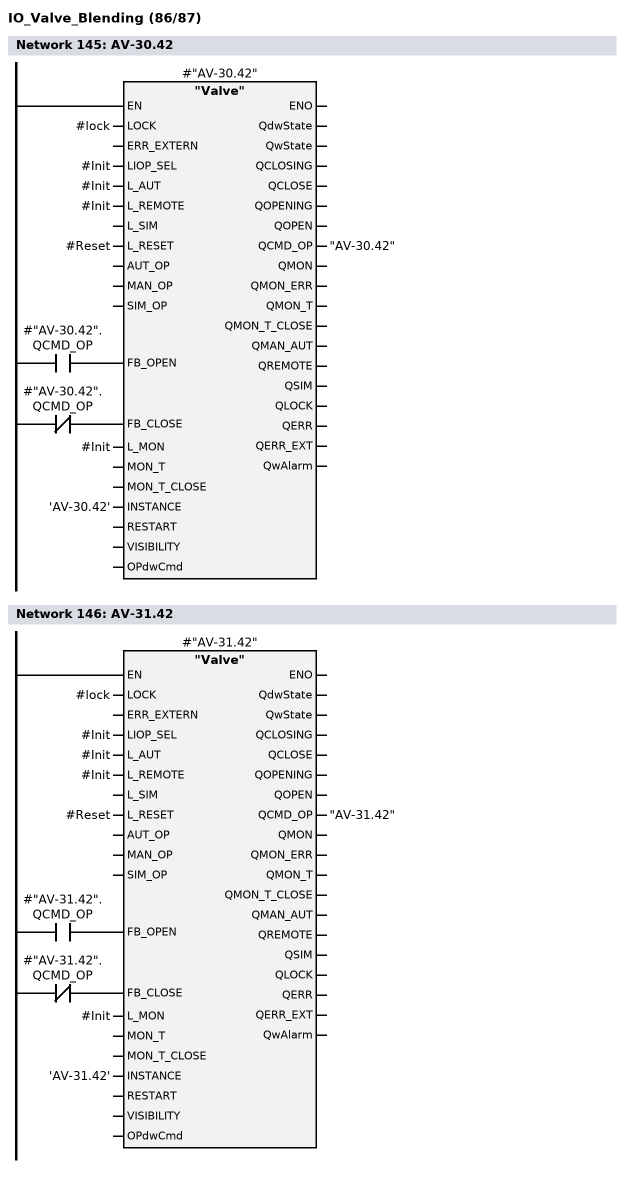
   RUNG wire#powerrail
      #"AV-30.42"(FB_OPEN := wire#w1, FB_CLOSE := wire#w2, LOCK := #lock, ERR_EXTERN :=, LIOP_SEL := #Init, L_AUT := #Init, L_REMOTE := #Init, L_SIM :=, L_RESET := #Reset, AUT_OP :=, MAN_OP :=, SIM_OP :=, L_MON := #Init, MON_T :=, MON_T_CLOSE :=, INSTANCE := 'AV-30.42', RESTART :=, VISIBILITY :=, OPdwCmd :=, QdwState =>, QwState =>, QCLOSING =>, QCLOSE =>, QOPENING =>, QOPEN =>, QCMD_OP => "AV-30.42", QMON =>, QMON_ERR =>, QMON_T =>, QMON_T_CLOSE =>, QMAN_AUT =>, QREMOTE =>, QSIM =>, QLOCK =>, QERR =>, QERR_EXT =>, QwAlarm =>)
   END_RUNG
   RUNG wire#powerrail
      Contact( #"AV-30.42".QCMD_OP )
   END_RUNG wire#w1
   RUNG wire#powerrail
      I_Contact( #"AV-30.42".QCMD_OP )
   END_RUNG wire#w2
   // the same network as SCL:
   #"AV-30.42"(LOCK := #lock,   // "Valve"
               LIOP_SEL := #Init,
               L_AUT := #Init,
               L_REMOTE := #Init,
               L_RESET := #Reset,
               FB_OPEN := #"AV-30.42".QCMD_OP,
               FB_CLOSE := NOT #"AV-30.42".QCMD_OP,
               L_MON := #Init,
               INSTANCE := 'AV-30.42',
               QCMD_OP => "AV-30.42");
END_REGION

REGION Network 146: AV-31.42
   RUNG wire#powerrail
      #"AV-31.42"(FB_OPEN := wire#w1, FB_CLOSE := wire#w2, LOCK := #lock, ERR_EXTERN :=, LIOP_SEL := #Init, L_AUT := #Init, L_REMOTE := #Init, L_SIM :=, L_RESET := #Reset, AUT_OP :=, MAN_OP :=, SIM_OP :=, L_MON := #Init, MON_T :=, MON_T_CLOSE :=, INSTANCE := 'AV-31.42', RESTART :=, VISIBILITY :=, OPdwCmd :=, QdwState =>, QwState =>, QCLOSING =>, QCLOSE =>, QOPENING =>, QOPEN =>, QCMD_OP => "AV-31.42", QMON =>, QMON_ERR =>, QMON_T =>, QMON_T_CLOSE =>, QMAN_AUT =>, QREMOTE =>, QSIM =>, QLOCK =>, QERR =>, QERR_EXT =>, QwAlarm =>)
   END_RUNG
   RUNG wire#powerrail
      Contact( #"AV-31.42".QCMD_OP )
   END_RUNG wire#w1
   RUNG wire#powerrail
      I_Contact( #"AV-31.42".QCMD_OP )
   END_RUNG wire#w2
   // the same network as SCL:
   #"AV-31.42"(LOCK := #lock,   // "Valve"
               LIOP_SEL := #Init,
               L_AUT := #Init,
               L_REMOTE := #Init,
               L_RESET := #Reset,
               FB_OPEN := #"AV-31.42".QCMD_OP,
               FB_CLOSE := NOT #"AV-31.42".QCMD_OP,
               L_MON := #Init,
               INSTANCE := 'AV-31.42',
               QCMD_OP => "AV-31.42");
END_REGION

REGION Network 147: AV-32.04
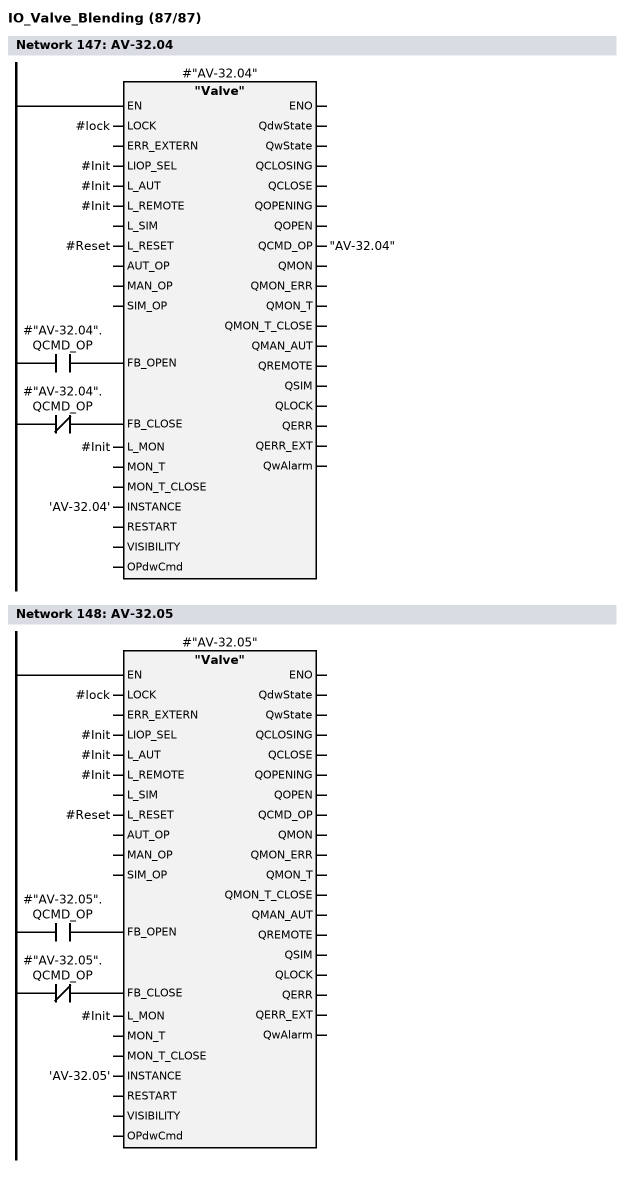
   RUNG wire#powerrail
      #"AV-32.04"(FB_OPEN := wire#w1, FB_CLOSE := wire#w2, LOCK := #lock, ERR_EXTERN :=, LIOP_SEL := #Init, L_AUT := #Init, L_REMOTE := #Init, L_SIM :=, L_RESET := #Reset, AUT_OP :=, MAN_OP :=, SIM_OP :=, L_MON := #Init, MON_T :=, MON_T_CLOSE :=, INSTANCE := 'AV-32.04', RESTART :=, VISIBILITY :=, OPdwCmd :=, QdwState =>, QwState =>, QCLOSING =>, QCLOSE =>, QOPENING =>, QOPEN =>, QCMD_OP => "AV-32.04", QMON =>, QMON_ERR =>, QMON_T =>, QMON_T_CLOSE =>, QMAN_AUT =>, QREMOTE =>, QSIM =>, QLOCK =>, QERR =>, QERR_EXT =>, QwAlarm =>)
   END_RUNG
   RUNG wire#powerrail
      Contact( #"AV-32.04".QCMD_OP )
   END_RUNG wire#w1
   RUNG wire#powerrail
      I_Contact( #"AV-32.04".QCMD_OP )
   END_RUNG wire#w2
   // the same network as SCL:
   #"AV-32.04"(LOCK := #lock,   // "Valve"
               LIOP_SEL := #Init,
               L_AUT := #Init,
               L_REMOTE := #Init,
               L_RESET := #Reset,
               FB_OPEN := #"AV-32.04".QCMD_OP,
               FB_CLOSE := NOT #"AV-32.04".QCMD_OP,
               L_MON := #Init,
               INSTANCE := 'AV-32.04',
               QCMD_OP => "AV-32.04");
END_REGION

REGION Network 148: AV-32.05
   RUNG wire#powerrail
      #"AV-32.05"(FB_OPEN := wire#w1, FB_CLOSE := wire#w2, LOCK := #lock, ERR_EXTERN :=, LIOP_SEL := #Init, L_AUT := #Init, L_REMOTE := #Init, L_SIM :=, L_RESET := #Reset, AUT_OP :=, MAN_OP :=, SIM_OP :=, L_MON := #Init, MON_T :=, MON_T_CLOSE :=, INSTANCE := 'AV-32.05', RESTART :=, VISIBILITY :=, OPdwCmd :=, QdwState =>, QwState =>, QCLOSING =>, QCLOSE =>, QOPENING =>, QOPEN =>, QCMD_OP =>, QMON =>, QMON_ERR =>, QMON_T =>, QMON_T_CLOSE =>, QMAN_AUT =>, QREMOTE =>, QSIM =>, QLOCK =>, QERR =>, QERR_EXT =>, QwAlarm =>)
   END_RUNG
   RUNG wire#powerrail
      Contact( #"AV-32.05".QCMD_OP )
   END_RUNG wire#w1
   RUNG wire#powerrail
      I_Contact( #"AV-32.05".QCMD_OP )
   END_RUNG wire#w2
   // the same network as SCL:
   #"AV-32.05"(LOCK := #lock,   // "Valve"
               LIOP_SEL := #Init,
               L_AUT := #Init,
               L_REMOTE := #Init,
               L_RESET := #Reset,
               FB_OPEN := #"AV-32.05".QCMD_OP,
               FB_CLOSE := NOT #"AV-32.05".QCMD_OP,
               L_MON := #Init,
               INSTANCE := 'AV-32.05');
END_REGION
END_FUNCTION_BLOCK

FUNCTION_BLOCK "IO Valve T01 HWT"   // FB301, LAD
{ S7_Optimized_Access := 'FALSE' }
VERSION : 0.1
// stored: AutoNumber false, IsIECCheckEnabled false, SetENOAutomatically false, UDAEnableTagReadback false
   VAR_INPUT
      lock : Bool;
      Init : Bool;
      Reset : Bool;
   END_VAR
   VAR
      "AV-01.01" { S7_SetPoint := 'True'} : "Valve";   // AUTO BUTTERFLY VALVE INLET HOT WATER CIRC. TO HOT WATER TANK T-01.00
      "AV-01.02" { S7_SetPoint := 'True'} : "Valve";   // AUTO BUTTERFLY VALVE INLET PROCESS WATER TO HOT WATER TANK T-01.00
      "AV-01.03" { S7_SetPoint := 'True'} : "Valve";   // AUTO BUTTERFLY VALVE CIP RETURN LINE 1
      "AV-01.04" { S7_SetPoint := 'True'} : "Valve";   // AUTO BUTTERFLY VALVE CIP SUPPLY HOT WATER TANK T-01.00
      "AV-01.05" { S7_SetPoint := 'True'} : "Valve";
      "AV-01.06" { S7_SetPoint := 'True'} : "Valve";
      "AV-01.07" { S7_SetPoint := 'True'} : "Valve";
      "AV-01.08" { S7_SetPoint := 'True'} : "Valve";
      "AV-01.09" { S7_SetPoint := 'True'} : "Valve";
      "AV-01.10" { S7_SetPoint := 'True'} : "Valve";   // AUTO ANGLE SEAT VALVE STEAM SUPPLY
      "AV-01.11" { S7_SetPoint := 'True'} : "Valve";
      "AV-01.12" { S7_SetPoint := 'True'} : "Valve";
      "AV-01.13" { S7_SetPoint := 'True'} : "Valve";
      "AV-01.14" { S7_SetPoint := 'True'} : "Valve";
      "AV-01.15" { S7_SetPoint := 'True'} : "Valve";
      "CV-01.01" { S7_SetPoint := 'True'} : "Valve";   // CONTROL VALVE STEAM FOR PHE PROCESS PHE-01.01
   END_VAR
BEGIN

REGION Network 1: AV-01.01
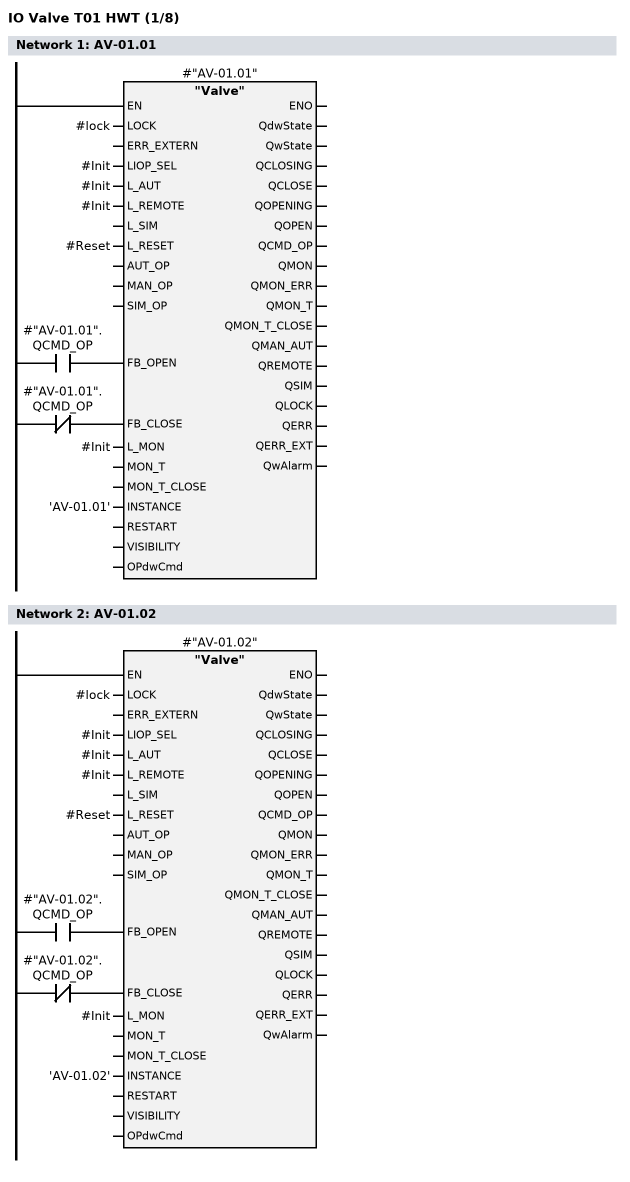
   RUNG wire#powerrail
      #"AV-01.01"(FB_OPEN := wire#w1, FB_CLOSE := wire#w2, LOCK := #lock, ERR_EXTERN :=, LIOP_SEL := #Init, L_AUT := #Init, L_REMOTE := #Init, L_SIM :=, L_RESET := #Reset, AUT_OP :=, MAN_OP :=, SIM_OP :=, L_MON := #Init, MON_T :=, MON_T_CLOSE :=, INSTANCE := 'AV-01.01', RESTART :=, VISIBILITY :=, OPdwCmd :=, QdwState =>, QwState =>, QCLOSING =>, QCLOSE =>, QOPENING =>, QOPEN =>, QCMD_OP =>, QMON =>, QMON_ERR =>, QMON_T =>, QMON_T_CLOSE =>, QMAN_AUT =>, QREMOTE =>, QSIM =>, QLOCK =>, QERR =>, QERR_EXT =>, QwAlarm =>)
   END_RUNG
   RUNG wire#powerrail
      Contact( #"AV-01.01".QCMD_OP )
   END_RUNG wire#w1
   RUNG wire#powerrail
      I_Contact( #"AV-01.01".QCMD_OP )
   END_RUNG wire#w2
   // the same network as SCL:
   #"AV-01.01"(LOCK := #lock,   // "Valve"
               LIOP_SEL := #Init,
               L_AUT := #Init,
               L_REMOTE := #Init,
               L_RESET := #Reset,
               FB_OPEN := #"AV-01.01".QCMD_OP,
               FB_CLOSE := NOT #"AV-01.01".QCMD_OP,
               L_MON := #Init,
               INSTANCE := 'AV-01.01');
END_REGION

REGION Network 2: AV-01.02
   RUNG wire#powerrail
      #"AV-01.02"(FB_OPEN := wire#w1, FB_CLOSE := wire#w2, LOCK := #lock, ERR_EXTERN :=, LIOP_SEL := #Init, L_AUT := #Init, L_REMOTE := #Init, L_SIM :=, L_RESET := #Reset, AUT_OP :=, MAN_OP :=, SIM_OP :=, L_MON := #Init, MON_T :=, MON_T_CLOSE :=, INSTANCE := 'AV-01.02', RESTART :=, VISIBILITY :=, OPdwCmd :=, QdwState =>, QwState =>, QCLOSING =>, QCLOSE =>, QOPENING =>, QOPEN =>, QCMD_OP =>, QMON =>, QMON_ERR =>, QMON_T =>, QMON_T_CLOSE =>, QMAN_AUT =>, QREMOTE =>, QSIM =>, QLOCK =>, QERR =>, QERR_EXT =>, QwAlarm =>)
   END_RUNG
   RUNG wire#powerrail
      Contact( #"AV-01.02".QCMD_OP )
   END_RUNG wire#w1
   RUNG wire#powerrail
      I_Contact( #"AV-01.02".QCMD_OP )
   END_RUNG wire#w2
   // the same network as SCL:
   #"AV-01.02"(LOCK := #lock,   // "Valve"
               LIOP_SEL := #Init,
               L_AUT := #Init,
               L_REMOTE := #Init,
               L_RESET := #Reset,
               FB_OPEN := #"AV-01.02".QCMD_OP,
               FB_CLOSE := NOT #"AV-01.02".QCMD_OP,
               L_MON := #Init,
               INSTANCE := 'AV-01.02');
END_REGION

REGION Network 3: AV-01.03
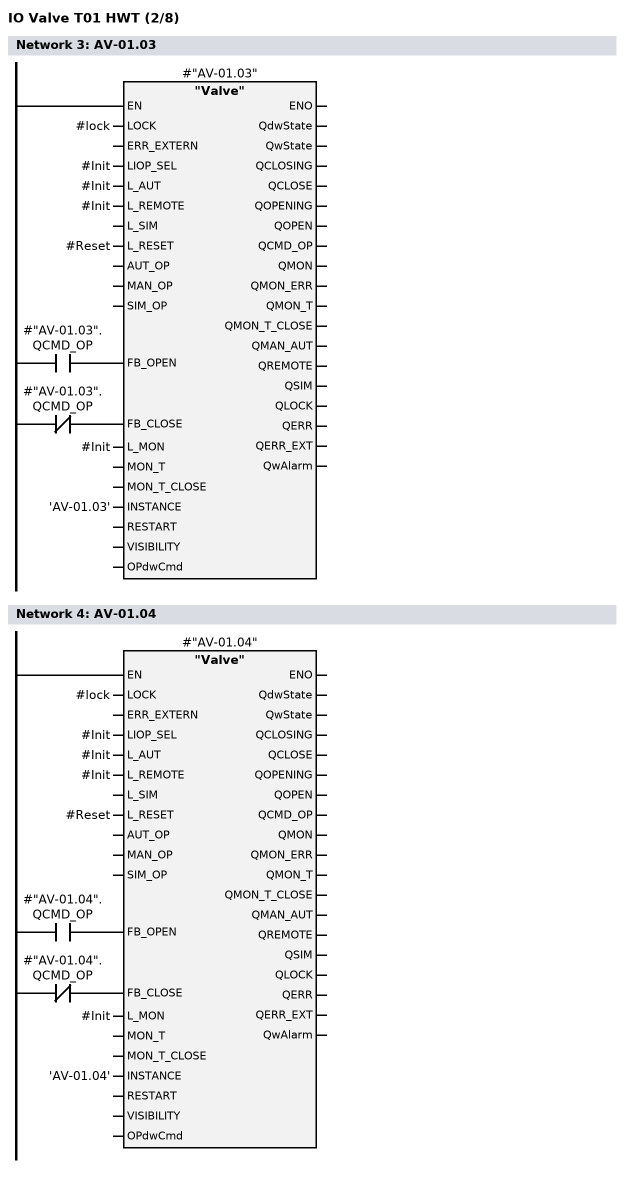
   RUNG wire#powerrail
      #"AV-01.03"(FB_OPEN := wire#w1, FB_CLOSE := wire#w2, LOCK := #lock, ERR_EXTERN :=, LIOP_SEL := #Init, L_AUT := #Init, L_REMOTE := #Init, L_SIM :=, L_RESET := #Reset, AUT_OP :=, MAN_OP :=, SIM_OP :=, L_MON := #Init, MON_T :=, MON_T_CLOSE :=, INSTANCE := 'AV-01.03', RESTART :=, VISIBILITY :=, OPdwCmd :=, QdwState =>, QwState =>, QCLOSING =>, QCLOSE =>, QOPENING =>, QOPEN =>, QCMD_OP =>, QMON =>, QMON_ERR =>, QMON_T =>, QMON_T_CLOSE =>, QMAN_AUT =>, QREMOTE =>, QSIM =>, QLOCK =>, QERR =>, QERR_EXT =>, QwAlarm =>)
   END_RUNG
   RUNG wire#powerrail
      Contact( #"AV-01.03".QCMD_OP )
   END_RUNG wire#w1
   RUNG wire#powerrail
      I_Contact( #"AV-01.03".QCMD_OP )
   END_RUNG wire#w2
   // the same network as SCL:
   #"AV-01.03"(LOCK := #lock,   // "Valve"
               LIOP_SEL := #Init,
               L_AUT := #Init,
               L_REMOTE := #Init,
               L_RESET := #Reset,
               FB_OPEN := #"AV-01.03".QCMD_OP,
               FB_CLOSE := NOT #"AV-01.03".QCMD_OP,
               L_MON := #Init,
               INSTANCE := 'AV-01.03');
END_REGION

REGION Network 4: AV-01.04
   RUNG wire#powerrail
      #"AV-01.04"(FB_OPEN := wire#w1, FB_CLOSE := wire#w2, LOCK := #lock, ERR_EXTERN :=, LIOP_SEL := #Init, L_AUT := #Init, L_REMOTE := #Init, L_SIM :=, L_RESET := #Reset, AUT_OP :=, MAN_OP :=, SIM_OP :=, L_MON := #Init, MON_T :=, MON_T_CLOSE :=, INSTANCE := 'AV-01.04', RESTART :=, VISIBILITY :=, OPdwCmd :=, QdwState =>, QwState =>, QCLOSING =>, QCLOSE =>, QOPENING =>, QOPEN =>, QCMD_OP =>, QMON =>, QMON_ERR =>, QMON_T =>, QMON_T_CLOSE =>, QMAN_AUT =>, QREMOTE =>, QSIM =>, QLOCK =>, QERR =>, QERR_EXT =>, QwAlarm =>)
   END_RUNG
   RUNG wire#powerrail
      Contact( #"AV-01.04".QCMD_OP )
   END_RUNG wire#w1
   RUNG wire#powerrail
      I_Contact( #"AV-01.04".QCMD_OP )
   END_RUNG wire#w2
   // the same network as SCL:
   #"AV-01.04"(LOCK := #lock,   // "Valve"
               LIOP_SEL := #Init,
               L_AUT := #Init,
               L_REMOTE := #Init,
               L_RESET := #Reset,
               FB_OPEN := #"AV-01.04".QCMD_OP,
               FB_CLOSE := NOT #"AV-01.04".QCMD_OP,
               L_MON := #Init,
               INSTANCE := 'AV-01.04');
END_REGION

REGION Network 5: AV-01.05
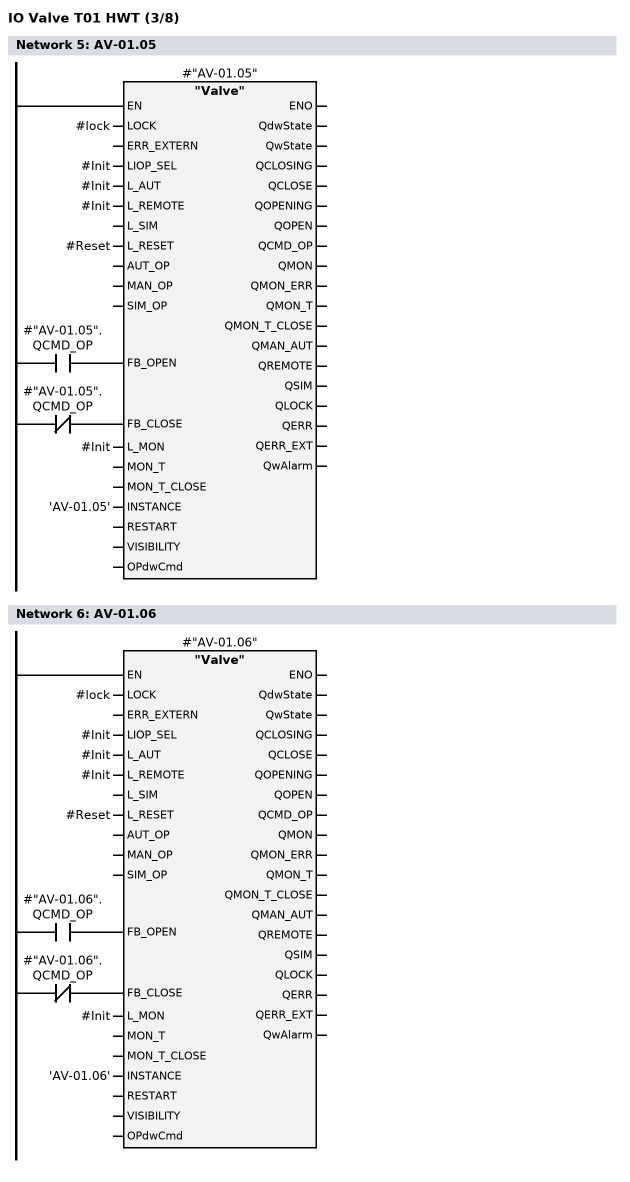
   RUNG wire#powerrail
      #"AV-01.05"(FB_OPEN := wire#w1, FB_CLOSE := wire#w2, LOCK := #lock, ERR_EXTERN :=, LIOP_SEL := #Init, L_AUT := #Init, L_REMOTE := #Init, L_SIM :=, L_RESET := #Reset, AUT_OP :=, MAN_OP :=, SIM_OP :=, L_MON := #Init, MON_T :=, MON_T_CLOSE :=, INSTANCE := 'AV-01.05', RESTART :=, VISIBILITY :=, OPdwCmd :=, QdwState =>, QwState =>, QCLOSING =>, QCLOSE =>, QOPENING =>, QOPEN =>, QCMD_OP =>, QMON =>, QMON_ERR =>, QMON_T =>, QMON_T_CLOSE =>, QMAN_AUT =>, QREMOTE =>, QSIM =>, QLOCK =>, QERR =>, QERR_EXT =>, QwAlarm =>)
   END_RUNG
   RUNG wire#powerrail
      Contact( #"AV-01.05".QCMD_OP )
   END_RUNG wire#w1
   RUNG wire#powerrail
      I_Contact( #"AV-01.05".QCMD_OP )
   END_RUNG wire#w2
   // the same network as SCL:
   #"AV-01.05"(LOCK := #lock,   // "Valve"
               LIOP_SEL := #Init,
               L_AUT := #Init,
               L_REMOTE := #Init,
               L_RESET := #Reset,
               FB_OPEN := #"AV-01.05".QCMD_OP,
               FB_CLOSE := NOT #"AV-01.05".QCMD_OP,
               L_MON := #Init,
               INSTANCE := 'AV-01.05');
END_REGION

REGION Network 6: AV-01.06
   RUNG wire#powerrail
      #"AV-01.06"(FB_OPEN := wire#w1, FB_CLOSE := wire#w2, LOCK := #lock, ERR_EXTERN :=, LIOP_SEL := #Init, L_AUT := #Init, L_REMOTE := #Init, L_SIM :=, L_RESET := #Reset, AUT_OP :=, MAN_OP :=, SIM_OP :=, L_MON := #Init, MON_T :=, MON_T_CLOSE :=, INSTANCE := 'AV-01.06', RESTART :=, VISIBILITY :=, OPdwCmd :=, QdwState =>, QwState =>, QCLOSING =>, QCLOSE =>, QOPENING =>, QOPEN =>, QCMD_OP =>, QMON =>, QMON_ERR =>, QMON_T =>, QMON_T_CLOSE =>, QMAN_AUT =>, QREMOTE =>, QSIM =>, QLOCK =>, QERR =>, QERR_EXT =>, QwAlarm =>)
   END_RUNG
   RUNG wire#powerrail
      Contact( #"AV-01.06".QCMD_OP )
   END_RUNG wire#w1
   RUNG wire#powerrail
      I_Contact( #"AV-01.06".QCMD_OP )
   END_RUNG wire#w2
   // the same network as SCL:
   #"AV-01.06"(LOCK := #lock,   // "Valve"
               LIOP_SEL := #Init,
               L_AUT := #Init,
               L_REMOTE := #Init,
               L_RESET := #Reset,
               FB_OPEN := #"AV-01.06".QCMD_OP,
               FB_CLOSE := NOT #"AV-01.06".QCMD_OP,
               L_MON := #Init,
               INSTANCE := 'AV-01.06');
END_REGION

REGION Network 7: AV-01.07
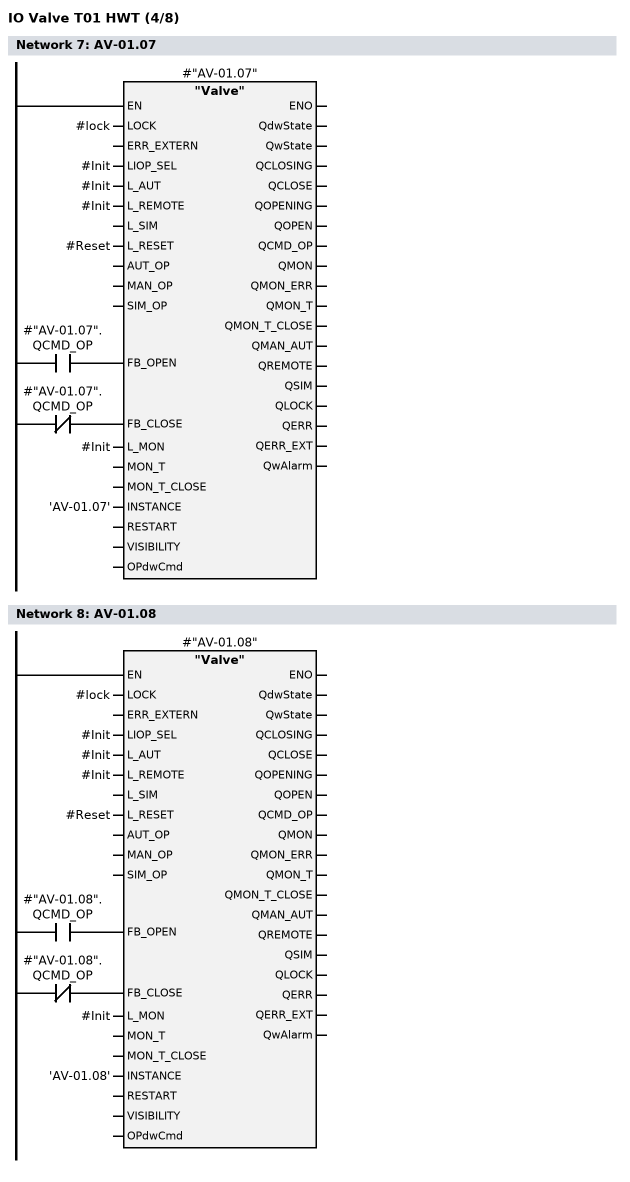
   RUNG wire#powerrail
      #"AV-01.07"(FB_OPEN := wire#w1, FB_CLOSE := wire#w2, LOCK := #lock, ERR_EXTERN :=, LIOP_SEL := #Init, L_AUT := #Init, L_REMOTE := #Init, L_SIM :=, L_RESET := #Reset, AUT_OP :=, MAN_OP :=, SIM_OP :=, L_MON := #Init, MON_T :=, MON_T_CLOSE :=, INSTANCE := 'AV-01.07', RESTART :=, VISIBILITY :=, OPdwCmd :=, QdwState =>, QwState =>, QCLOSING =>, QCLOSE =>, QOPENING =>, QOPEN =>, QCMD_OP =>, QMON =>, QMON_ERR =>, QMON_T =>, QMON_T_CLOSE =>, QMAN_AUT =>, QREMOTE =>, QSIM =>, QLOCK =>, QERR =>, QERR_EXT =>, QwAlarm =>)
   END_RUNG
   RUNG wire#powerrail
      Contact( #"AV-01.07".QCMD_OP )
   END_RUNG wire#w1
   RUNG wire#powerrail
      I_Contact( #"AV-01.07".QCMD_OP )
   END_RUNG wire#w2
   // the same network as SCL:
   #"AV-01.07"(LOCK := #lock,   // "Valve"
               LIOP_SEL := #Init,
               L_AUT := #Init,
               L_REMOTE := #Init,
               L_RESET := #Reset,
               FB_OPEN := #"AV-01.07".QCMD_OP,
               FB_CLOSE := NOT #"AV-01.07".QCMD_OP,
               L_MON := #Init,
               INSTANCE := 'AV-01.07');
END_REGION

REGION Network 8: AV-01.08
   RUNG wire#powerrail
      #"AV-01.08"(FB_OPEN := wire#w1, FB_CLOSE := wire#w2, LOCK := #lock, ERR_EXTERN :=, LIOP_SEL := #Init, L_AUT := #Init, L_REMOTE := #Init, L_SIM :=, L_RESET := #Reset, AUT_OP :=, MAN_OP :=, SIM_OP :=, L_MON := #Init, MON_T :=, MON_T_CLOSE :=, INSTANCE := 'AV-01.08', RESTART :=, VISIBILITY :=, OPdwCmd :=, QdwState =>, QwState =>, QCLOSING =>, QCLOSE =>, QOPENING =>, QOPEN =>, QCMD_OP =>, QMON =>, QMON_ERR =>, QMON_T =>, QMON_T_CLOSE =>, QMAN_AUT =>, QREMOTE =>, QSIM =>, QLOCK =>, QERR =>, QERR_EXT =>, QwAlarm =>)
   END_RUNG
   RUNG wire#powerrail
      Contact( #"AV-01.08".QCMD_OP )
   END_RUNG wire#w1
   RUNG wire#powerrail
      I_Contact( #"AV-01.08".QCMD_OP )
   END_RUNG wire#w2
   // the same network as SCL:
   #"AV-01.08"(LOCK := #lock,   // "Valve"
               LIOP_SEL := #Init,
               L_AUT := #Init,
               L_REMOTE := #Init,
               L_RESET := #Reset,
               FB_OPEN := #"AV-01.08".QCMD_OP,
               FB_CLOSE := NOT #"AV-01.08".QCMD_OP,
               L_MON := #Init,
               INSTANCE := 'AV-01.08');
END_REGION

REGION Network 9: AV-01.09
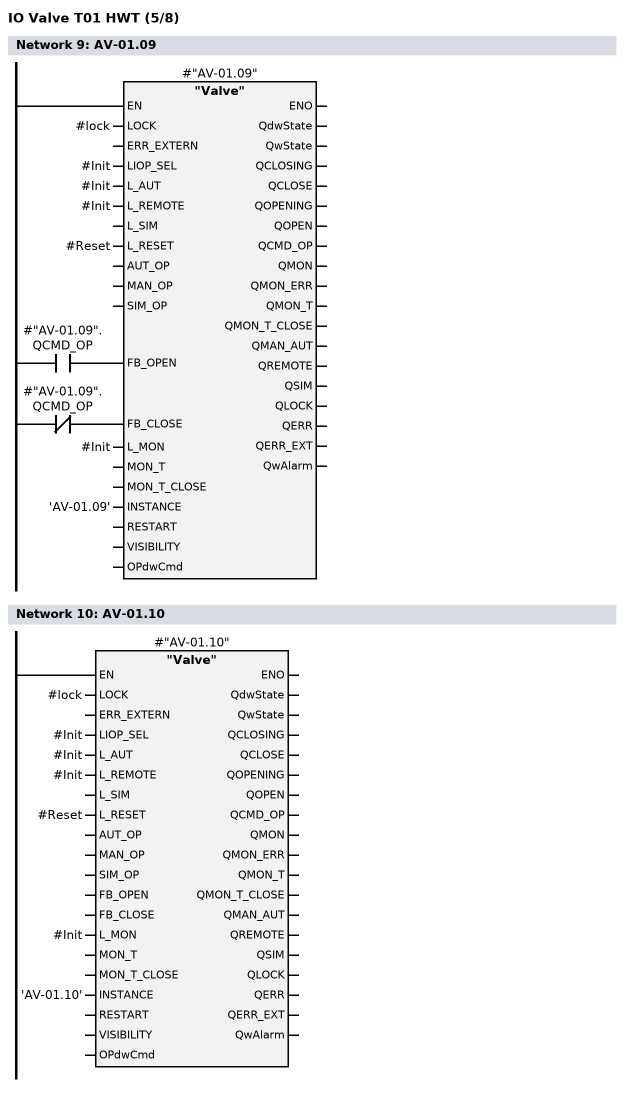
   RUNG wire#powerrail
      #"AV-01.09"(FB_OPEN := wire#w1, FB_CLOSE := wire#w2, LOCK := #lock, ERR_EXTERN :=, LIOP_SEL := #Init, L_AUT := #Init, L_REMOTE := #Init, L_SIM :=, L_RESET := #Reset, AUT_OP :=, MAN_OP :=, SIM_OP :=, L_MON := #Init, MON_T :=, MON_T_CLOSE :=, INSTANCE := 'AV-01.09', RESTART :=, VISIBILITY :=, OPdwCmd :=, QdwState =>, QwState =>, QCLOSING =>, QCLOSE =>, QOPENING =>, QOPEN =>, QCMD_OP =>, QMON =>, QMON_ERR =>, QMON_T =>, QMON_T_CLOSE =>, QMAN_AUT =>, QREMOTE =>, QSIM =>, QLOCK =>, QERR =>, QERR_EXT =>, QwAlarm =>)
   END_RUNG
   RUNG wire#powerrail
      Contact( #"AV-01.09".QCMD_OP )
   END_RUNG wire#w1
   RUNG wire#powerrail
      I_Contact( #"AV-01.09".QCMD_OP )
   END_RUNG wire#w2
   // the same network as SCL:
   #"AV-01.09"(LOCK := #lock,   // "Valve"
               LIOP_SEL := #Init,
               L_AUT := #Init,
               L_REMOTE := #Init,
               L_RESET := #Reset,
               FB_OPEN := #"AV-01.09".QCMD_OP,
               FB_CLOSE := NOT #"AV-01.09".QCMD_OP,
               L_MON := #Init,
               INSTANCE := 'AV-01.09');
END_REGION

REGION Network 10: AV-01.10
   RUNG wire#powerrail
      #"AV-01.10"(LOCK := #lock, ERR_EXTERN :=, LIOP_SEL := #Init, L_AUT := #Init, L_REMOTE := #Init, L_SIM :=, L_RESET := #Reset, AUT_OP :=, MAN_OP :=, SIM_OP :=, FB_OPEN :=, FB_CLOSE :=, L_MON := #Init, MON_T :=, MON_T_CLOSE :=, INSTANCE := 'AV-01.10', RESTART :=, VISIBILITY :=, OPdwCmd :=, QdwState =>, QwState =>, QCLOSING =>, QCLOSE =>, QOPENING =>, QOPEN =>, QCMD_OP =>, QMON =>, QMON_ERR =>, QMON_T =>, QMON_T_CLOSE =>, QMAN_AUT =>, QREMOTE =>, QSIM =>, QLOCK =>, QERR =>, QERR_EXT =>, QwAlarm =>)
   END_RUNG
   // the same network as SCL:
   #"AV-01.10"(LOCK := #lock,   // "Valve"
               LIOP_SEL := #Init,
               L_AUT := #Init,
               L_REMOTE := #Init,
               L_RESET := #Reset,
               L_MON := #Init,
               INSTANCE := 'AV-01.10');
END_REGION

REGION Network 11: AV-01.11
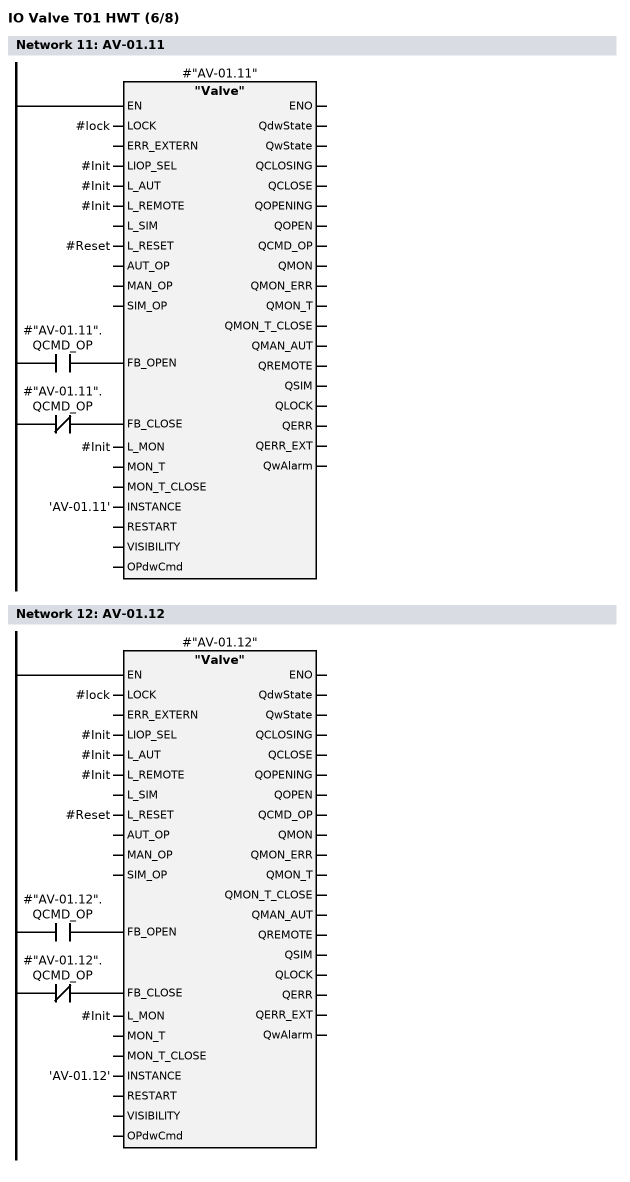
   RUNG wire#powerrail
      #"AV-01.11"(FB_OPEN := wire#w1, FB_CLOSE := wire#w2, LOCK := #lock, ERR_EXTERN :=, LIOP_SEL := #Init, L_AUT := #Init, L_REMOTE := #Init, L_SIM :=, L_RESET := #Reset, AUT_OP :=, MAN_OP :=, SIM_OP :=, L_MON := #Init, MON_T :=, MON_T_CLOSE :=, INSTANCE := 'AV-01.11', RESTART :=, VISIBILITY :=, OPdwCmd :=, QdwState =>, QwState =>, QCLOSING =>, QCLOSE =>, QOPENING =>, QOPEN =>, QCMD_OP =>, QMON =>, QMON_ERR =>, QMON_T =>, QMON_T_CLOSE =>, QMAN_AUT =>, QREMOTE =>, QSIM =>, QLOCK =>, QERR =>, QERR_EXT =>, QwAlarm =>)
   END_RUNG
   RUNG wire#powerrail
      Contact( #"AV-01.11".QCMD_OP )
   END_RUNG wire#w1
   RUNG wire#powerrail
      I_Contact( #"AV-01.11".QCMD_OP )
   END_RUNG wire#w2
   // the same network as SCL:
   #"AV-01.11"(LOCK := #lock,   // "Valve"
               LIOP_SEL := #Init,
               L_AUT := #Init,
               L_REMOTE := #Init,
               L_RESET := #Reset,
               FB_OPEN := #"AV-01.11".QCMD_OP,
               FB_CLOSE := NOT #"AV-01.11".QCMD_OP,
               L_MON := #Init,
               INSTANCE := 'AV-01.11');
END_REGION

REGION Network 12: AV-01.12
   RUNG wire#powerrail
      #"AV-01.12"(FB_OPEN := wire#w1, FB_CLOSE := wire#w2, LOCK := #lock, ERR_EXTERN :=, LIOP_SEL := #Init, L_AUT := #Init, L_REMOTE := #Init, L_SIM :=, L_RESET := #Reset, AUT_OP :=, MAN_OP :=, SIM_OP :=, L_MON := #Init, MON_T :=, MON_T_CLOSE :=, INSTANCE := 'AV-01.12', RESTART :=, VISIBILITY :=, OPdwCmd :=, QdwState =>, QwState =>, QCLOSING =>, QCLOSE =>, QOPENING =>, QOPEN =>, QCMD_OP =>, QMON =>, QMON_ERR =>, QMON_T =>, QMON_T_CLOSE =>, QMAN_AUT =>, QREMOTE =>, QSIM =>, QLOCK =>, QERR =>, QERR_EXT =>, QwAlarm =>)
   END_RUNG
   RUNG wire#powerrail
      Contact( #"AV-01.12".QCMD_OP )
   END_RUNG wire#w1
   RUNG wire#powerrail
      I_Contact( #"AV-01.12".QCMD_OP )
   END_RUNG wire#w2
   // the same network as SCL:
   #"AV-01.12"(LOCK := #lock,   // "Valve"
               LIOP_SEL := #Init,
               L_AUT := #Init,
               L_REMOTE := #Init,
               L_RESET := #Reset,
               FB_OPEN := #"AV-01.12".QCMD_OP,
               FB_CLOSE := NOT #"AV-01.12".QCMD_OP,
               L_MON := #Init,
               INSTANCE := 'AV-01.12');
END_REGION

REGION Network 13: AV-01.13
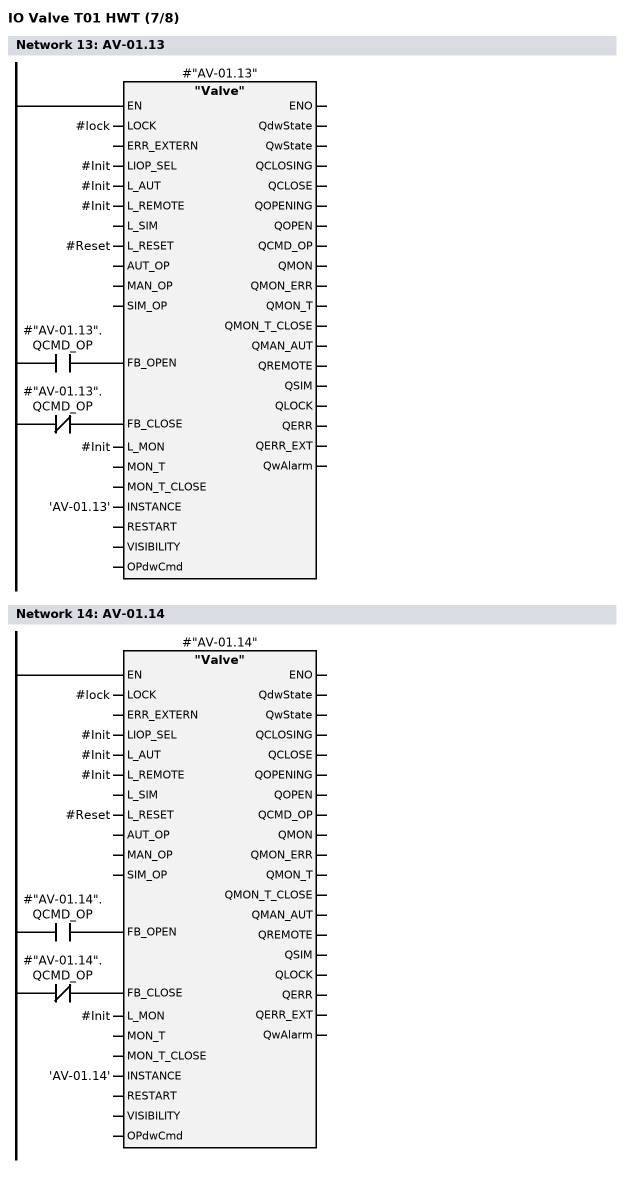
   RUNG wire#powerrail
      #"AV-01.13"(FB_OPEN := wire#w1, FB_CLOSE := wire#w2, LOCK := #lock, ERR_EXTERN :=, LIOP_SEL := #Init, L_AUT := #Init, L_REMOTE := #Init, L_SIM :=, L_RESET := #Reset, AUT_OP :=, MAN_OP :=, SIM_OP :=, L_MON := #Init, MON_T :=, MON_T_CLOSE :=, INSTANCE := 'AV-01.13', RESTART :=, VISIBILITY :=, OPdwCmd :=, QdwState =>, QwState =>, QCLOSING =>, QCLOSE =>, QOPENING =>, QOPEN =>, QCMD_OP =>, QMON =>, QMON_ERR =>, QMON_T =>, QMON_T_CLOSE =>, QMAN_AUT =>, QREMOTE =>, QSIM =>, QLOCK =>, QERR =>, QERR_EXT =>, QwAlarm =>)
   END_RUNG
   RUNG wire#powerrail
      Contact( #"AV-01.13".QCMD_OP )
   END_RUNG wire#w1
   RUNG wire#powerrail
      I_Contact( #"AV-01.13".QCMD_OP )
   END_RUNG wire#w2
   // the same network as SCL:
   #"AV-01.13"(LOCK := #lock,   // "Valve"
               LIOP_SEL := #Init,
               L_AUT := #Init,
               L_REMOTE := #Init,
               L_RESET := #Reset,
               FB_OPEN := #"AV-01.13".QCMD_OP,
               FB_CLOSE := NOT #"AV-01.13".QCMD_OP,
               L_MON := #Init,
               INSTANCE := 'AV-01.13');
END_REGION

REGION Network 14: AV-01.14
   RUNG wire#powerrail
      #"AV-01.14"(FB_OPEN := wire#w1, FB_CLOSE := wire#w2, LOCK := #lock, ERR_EXTERN :=, LIOP_SEL := #Init, L_AUT := #Init, L_REMOTE := #Init, L_SIM :=, L_RESET := #Reset, AUT_OP :=, MAN_OP :=, SIM_OP :=, L_MON := #Init, MON_T :=, MON_T_CLOSE :=, INSTANCE := 'AV-01.14', RESTART :=, VISIBILITY :=, OPdwCmd :=, QdwState =>, QwState =>, QCLOSING =>, QCLOSE =>, QOPENING =>, QOPEN =>, QCMD_OP =>, QMON =>, QMON_ERR =>, QMON_T =>, QMON_T_CLOSE =>, QMAN_AUT =>, QREMOTE =>, QSIM =>, QLOCK =>, QERR =>, QERR_EXT =>, QwAlarm =>)
   END_RUNG
   RUNG wire#powerrail
      Contact( #"AV-01.14".QCMD_OP )
   END_RUNG wire#w1
   RUNG wire#powerrail
      I_Contact( #"AV-01.14".QCMD_OP )
   END_RUNG wire#w2
   // the same network as SCL:
   #"AV-01.14"(LOCK := #lock,   // "Valve"
               LIOP_SEL := #Init,
               L_AUT := #Init,
               L_REMOTE := #Init,
               L_RESET := #Reset,
               FB_OPEN := #"AV-01.14".QCMD_OP,
               FB_CLOSE := NOT #"AV-01.14".QCMD_OP,
               L_MON := #Init,
               INSTANCE := 'AV-01.14');
END_REGION

REGION Network 15: AV-01.15
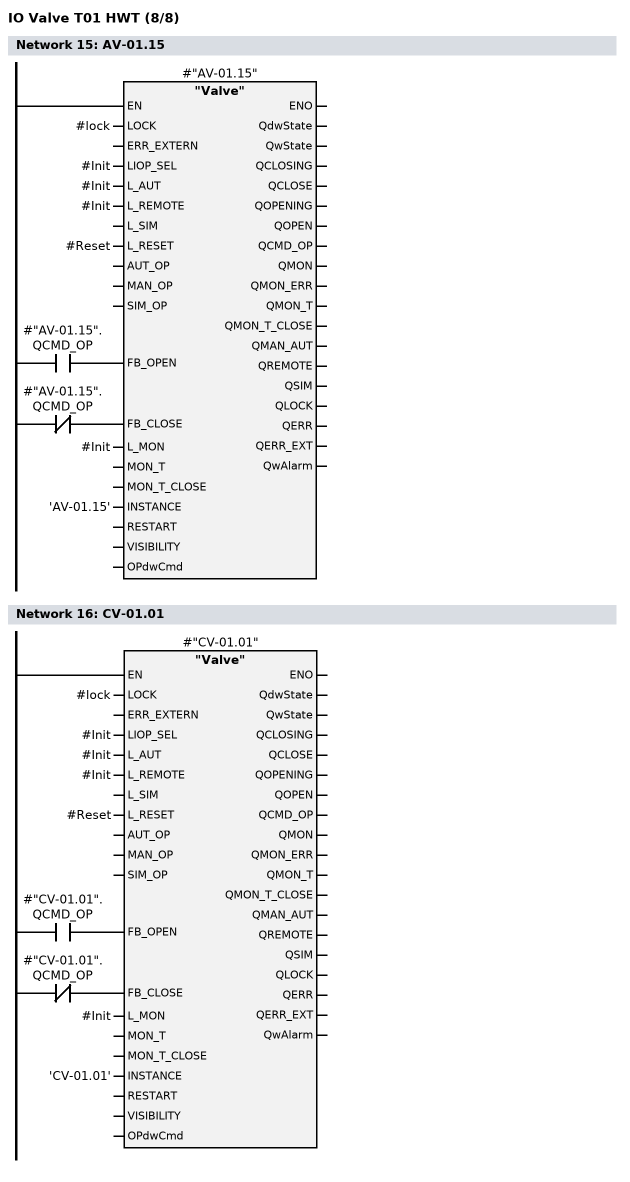
   RUNG wire#powerrail
      #"AV-01.15"(FB_OPEN := wire#w1, FB_CLOSE := wire#w2, LOCK := #lock, ERR_EXTERN :=, LIOP_SEL := #Init, L_AUT := #Init, L_REMOTE := #Init, L_SIM :=, L_RESET := #Reset, AUT_OP :=, MAN_OP :=, SIM_OP :=, L_MON := #Init, MON_T :=, MON_T_CLOSE :=, INSTANCE := 'AV-01.15', RESTART :=, VISIBILITY :=, OPdwCmd :=, QdwState =>, QwState =>, QCLOSING =>, QCLOSE =>, QOPENING =>, QOPEN =>, QCMD_OP =>, QMON =>, QMON_ERR =>, QMON_T =>, QMON_T_CLOSE =>, QMAN_AUT =>, QREMOTE =>, QSIM =>, QLOCK =>, QERR =>, QERR_EXT =>, QwAlarm =>)
   END_RUNG
   RUNG wire#powerrail
      Contact( #"AV-01.15".QCMD_OP )
   END_RUNG wire#w1
   RUNG wire#powerrail
      I_Contact( #"AV-01.15".QCMD_OP )
   END_RUNG wire#w2
   // the same network as SCL:
   #"AV-01.15"(LOCK := #lock,   // "Valve"
               LIOP_SEL := #Init,
               L_AUT := #Init,
               L_REMOTE := #Init,
               L_RESET := #Reset,
               FB_OPEN := #"AV-01.15".QCMD_OP,
               FB_CLOSE := NOT #"AV-01.15".QCMD_OP,
               L_MON := #Init,
               INSTANCE := 'AV-01.15');
END_REGION

REGION Network 16: CV-01.01
   RUNG wire#powerrail
      #"CV-01.01"(FB_OPEN := wire#w1, FB_CLOSE := wire#w2, LOCK := #lock, ERR_EXTERN :=, LIOP_SEL := #Init, L_AUT := #Init, L_REMOTE := #Init, L_SIM :=, L_RESET := #Reset, AUT_OP :=, MAN_OP :=, SIM_OP :=, L_MON := #Init, MON_T :=, MON_T_CLOSE :=, INSTANCE := 'CV-01.01', RESTART :=, VISIBILITY :=, OPdwCmd :=, QdwState =>, QwState =>, QCLOSING =>, QCLOSE =>, QOPENING =>, QOPEN =>, QCMD_OP =>, QMON =>, QMON_ERR =>, QMON_T =>, QMON_T_CLOSE =>, QMAN_AUT =>, QREMOTE =>, QSIM =>, QLOCK =>, QERR =>, QERR_EXT =>, QwAlarm =>)
   END_RUNG
   RUNG wire#powerrail
      Contact( #"CV-01.01".QCMD_OP )
   END_RUNG wire#w1
   RUNG wire#powerrail
      I_Contact( #"CV-01.01".QCMD_OP )
   END_RUNG wire#w2
   // the same network as SCL:
   #"CV-01.01"(LOCK := #lock,   // "Valve"
               LIOP_SEL := #Init,
               L_AUT := #Init,
               L_REMOTE := #Init,
               L_RESET := #Reset,
               FB_OPEN := #"CV-01.01".QCMD_OP,
               FB_CLOSE := NOT #"CV-01.01".QCMD_OP,
               L_MON := #Init,
               INSTANCE := 'CV-01.01');
END_REGION
END_FUNCTION_BLOCK

FUNCTION_BLOCK "BLEND"   // FB16, LAD
{ S7_Optimized_Access := 'FALSE' }
VERSION : 0.1
// stored: AutoNumber true, IsIECCheckEnabled false, SetENOAutomatically false, UDAEnableTagReadback false
   VAR_INPUT
      Lock : Bool := true;
      Reset : Bool;
      ENTransfer : Bool;
      ENProd : Bool;
      THE_ProdReq : Bool;   // THE Product Request
      THE_ProdLineOpen : Bool;   // THE Line Transfer Open
      THE_CIPLineOpen : Bool;   // THE CIP Line Open
      THE_CIP_En : Bool;   // THE CIP Enable
      MixproofFlip : Bool;
      FB_AV_Transfer : Bool;
      FB_P_Transfer : Bool;
      Level : Real;   // Tank Level Transmitter
      Temp : Real;   // Tank Temp Transmitter
      TransfPump_AVSpeed : Real;
   END_VAR
   VAR_OUTPUT
      Q_Prod : Bool;   // Product Available
      Q_Trans : Bool;   // Transfer to Mix in Progress
      Q_CIPReq : Bool;   // CIP Request
      Q_MixProofFlif : Bool;   // Mixproof Valve Flip
      QAV_Transfer : Bool;
      QP_Transfer : Bool;
   END_VAR
   VAR DB_SPECIFIC
      Cmd : Struct
         Transfer_ON : Bool;
         Transfer_OFF : Bool;
      END_STRUCT;
      HMI : Struct
         Cmd : DWord;
         Cmd_EN : DWord;
         Cmd_Stat : DWord;
         MatSel : DWord;
         DoseStart : DWord;
         DosePause : DWord;
         DoseStop : DWord;
         DoseState : DWord;
      END_STRUCT;
      Tank_Par : Struct
         LL : Real := 2.0;   // Tank Low Level
         LB_OFF : Real := 17.0;
         LB_ON : Real := 20.0;
         LB1_OFF : Real := 10.0;   // Level Under Lower Blade
         LB1_ON : Real := 15.0;   // Level Over Lower Blade
         LB2_OFF : Real := 30.0;   // Level Under Medium Blade
         LB2_ON : Real := 35.0;   // Level Over Medium Blade
         LB3_OFF : Real := 60.0;   // Level Under Upper Blade
         LB3_ON : Real := 65.0;   // Level Over Upper Blade
         P01_ProdSP : Real := 5.0;   // Transfer pump Setpoint speed at product transfer
         P01_CIPSP : Real := 50.0;   // Transfer pump Setpoint speed at CIP
      END_STRUCT;
      Tank_Sta : Struct   // Tank Low Level
         LL : Bool;   // Level Under Lower Blade
         LB_OFF : Bool;
         LB_ON : Bool;
         LB1_OFF : Bool;   // Level Over Lower Blade
         LB1_ON : Bool;   // Level Under Medium Blade
         LB2_OFF : Bool;   // Level Over Medium Blade
         LB2_ON : Bool;   // Level Under Upper Blade
         LB3_OFF : Bool;   // Level Over Upper Blade
         LB3_ON : Bool;
         Agi_ON : Bool;
         TranferON : Bool;
         Inload : Bool;
         CIPRequest : Bool;
         AwysON : Bool;
      END_STRUCT;
   END_VAR
   VAR
      SP_Water : "RawDose";
      SP_Sugar { S7_SetPoint := 'True'} : "RawDose";
      SP_Garam { S7_SetPoint := 'True'} : "RawDose";
      SP_ChiliAwet_1 { S7_SetPoint := 'True'} : "RawDose";
      SP_ChiliAwet_2 { S7_SetPoint := 'True'} : "RawDose";
      SP_ChiliAwet_3 { S7_SetPoint := 'True'} : "RawDose";
      SP_ChiliFresh_1 { S7_SetPoint := 'True'} : "RawDose";
      SP_ChiliFresh_2 { S7_SetPoint := 'True'} : "RawDose";
      SP_ChiliFresh_3 { S7_SetPoint := 'True'} : "RawDose";
      SP_Garlic { S7_SetPoint := 'True'} : "RawDose";
      SP_Vinegar { S7_SetPoint := 'True'} : "RawDose";
      SP_Tomato { S7_SetPoint := 'True'} : "RawDose";
      SP_Homomix { S7_SetPoint := 'True'} : "RawDose";
      SP_Rework { S7_SetPoint := 'True'} : "RawDose";
      Water : "DOSE";
      Sugar { S7_SetPoint := 'True'} : "DOSE";
      Garam : "DOSE";
      ChiliAwet_1 { S7_SetPoint := 'True'} : "DOSE";
      ChiliAwet_2 { S7_SetPoint := 'True'} : "DOSE";
      ChiliAwet_3 { S7_SetPoint := 'True'} : "DOSE";
      ChiliFresh_1 { S7_SetPoint := 'True'} : "DOSE";
      ChiliFresh_2 { S7_SetPoint := 'True'} : "DOSE";
      ChiliFresh_3 { S7_SetPoint := 'True'} : "DOSE";
      Garlic { S7_SetPoint := 'True'} : "DOSE";
      Vinegar { S7_SetPoint := 'True'} : "DOSE";
      Tomato { S7_SetPoint := 'True'} : "DOSE";
      Homomix { S7_SetPoint := 'True'} : "DOSE";
      Rework { S7_SetPoint := 'True'} : "DOSE";
   END_VAR
   VAR DB_SPECIFIC
      RdyforTransfer : Struct
         cmd_on : Bool;
         cmd_off : Bool;
         EnCmd : Bool;
         Stat_ON : Bool;
         Stat_Stop : Bool;
      END_STRUCT;
      Transfer : Struct
         cmd_on : Bool;
         cmd_off : Bool;
         EnCmd : Bool;
         Stat_ON : Bool;
         Stat_Stop : Bool;
      END_STRUCT;
      CIP : Struct
         cmd_on : Bool;
         cmd_off : Bool;
         EnCmd : Bool;
         Stat_ON : Bool;
         Stat_Stop : Bool;
      END_STRUCT;
      Agitator : Struct
         cmd_on : Bool;
         cmd_off : Bool;
         EnCmd : Bool;
         Stat_ON : Bool;
         Stat_Stop : Bool;
      END_STRUCT;
      PumpOFFTimer : TON_TIME;
      TransitionTimer { S7_SetPoint := 'True'} : TON_TIME;
   END_VAR
BEGIN

REGION Network 1: Always ON
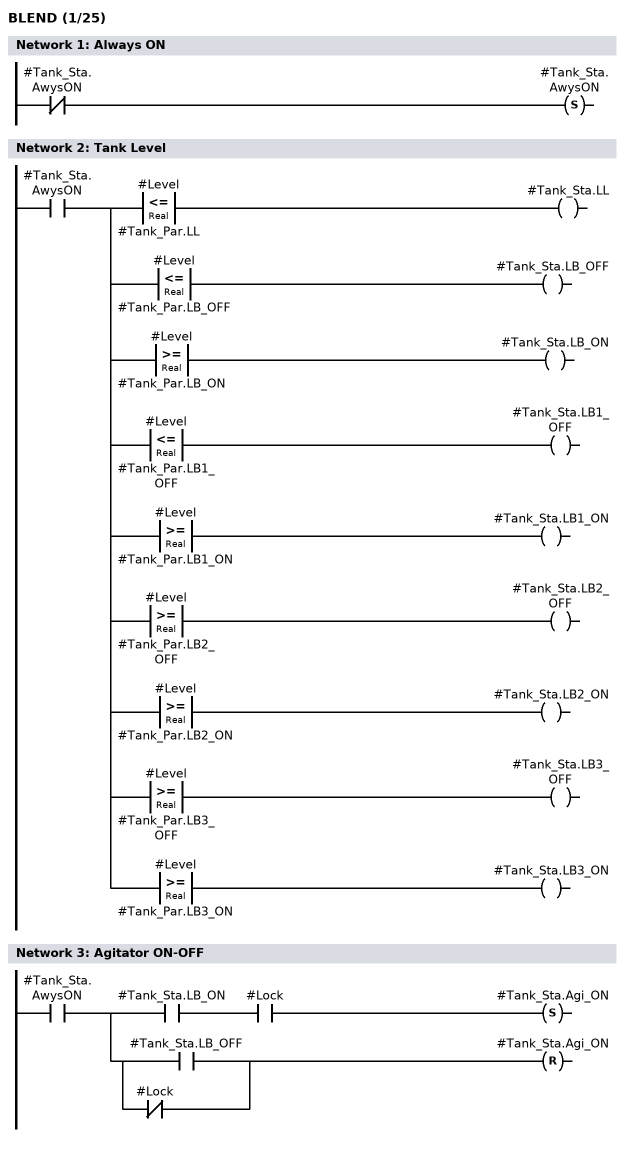
   RUNG wire#powerrail
      I_Contact( #Tank_Sta.AwysON )
      S_Coil( #Tank_Sta.AwysON )
   END_RUNG
   // the same network as SCL:
   IF NOT #Tank_Sta.AwysON THEN #Tank_Sta.AwysON := TRUE; END_IF;
END_REGION

REGION Network 2: Tank Level
   RUNG wire#powerrail
      Contact( #Tank_Sta.AwysON )
      wire#w1
      { S7_Templates := "SrcType := Real" } LE_Contact(in1 := #Level, in2 := #Tank_Par.LL)
      Coil( #Tank_Sta.LL )
   END_RUNG
   RUNG wire#w1
      { S7_Templates := "SrcType := Real" } LE_Contact(in1 := #Level, in2 := #Tank_Par.LB_OFF)
      Coil( #Tank_Sta.LB_OFF )
   END_RUNG
   RUNG wire#w1
      { S7_Templates := "SrcType := Real" } GE_Contact(in1 := #Level, in2 := #Tank_Par.LB_ON)
      Coil( #Tank_Sta.LB_ON )
   END_RUNG
   RUNG wire#w1
      { S7_Templates := "SrcType := Real" } LE_Contact(in1 := #Level, in2 := #Tank_Par.LB1_OFF)
      Coil( #Tank_Sta.LB1_OFF )
   END_RUNG
   RUNG wire#w1
      { S7_Templates := "SrcType := Real" } GE_Contact(in1 := #Level, in2 := #Tank_Par.LB1_ON)
      Coil( #Tank_Sta.LB1_ON )
   END_RUNG
   RUNG wire#w1
      { S7_Templates := "SrcType := Real" } GE_Contact(in1 := #Level, in2 := #Tank_Par.LB2_OFF)
      Coil( #Tank_Sta.LB2_OFF )
   END_RUNG
   RUNG wire#w1
      { S7_Templates := "SrcType := Real" } GE_Contact(in1 := #Level, in2 := #Tank_Par.LB2_ON)
      Coil( #Tank_Sta.LB2_ON )
   END_RUNG
   RUNG wire#w1
      { S7_Templates := "SrcType := Real" } GE_Contact(in1 := #Level, in2 := #Tank_Par.LB3_OFF)
      Coil( #Tank_Sta.LB3_OFF )
   END_RUNG
   RUNG wire#w1
      { S7_Templates := "SrcType := Real" } GE_Contact(in1 := #Level, in2 := #Tank_Par.LB3_ON)
      Coil( #Tank_Sta.LB3_ON )
   END_RUNG
   // the same network as SCL:
   #Tank_Sta.LL := #Tank_Sta.AwysON AND (#Level <= #Tank_Par.LL);
   #Tank_Sta.LB_OFF := #Tank_Sta.AwysON AND (#Level <= #Tank_Par.LB_OFF);
   #Tank_Sta.LB_ON := #Tank_Sta.AwysON AND (#Level >= #Tank_Par.LB_ON);
   #Tank_Sta.LB1_OFF := #Tank_Sta.AwysON AND (#Level <= #Tank_Par.LB1_OFF);
   #Tank_Sta.LB1_ON := #Tank_Sta.AwysON AND (#Level >= #Tank_Par.LB1_ON);
   #Tank_Sta.LB2_OFF := #Tank_Sta.AwysON AND (#Level >= #Tank_Par.LB2_OFF);
   #Tank_Sta.LB2_ON := #Tank_Sta.AwysON AND (#Level >= #Tank_Par.LB2_ON);
   #Tank_Sta.LB3_OFF := #Tank_Sta.AwysON AND (#Level >= #Tank_Par.LB3_OFF);
   #Tank_Sta.LB3_ON := #Tank_Sta.AwysON AND (#Level >= #Tank_Par.LB3_ON);
END_REGION

REGION Network 3: Agitator ON-OFF
   RUNG wire#powerrail
      Contact( #Tank_Sta.AwysON )
      wire#w1
      Contact( #Tank_Sta.LB_ON )
      Contact( #Lock )
      S_Coil( #Tank_Sta.Agi_ON )
   END_RUNG
   RUNG wire#w1
      Contact( #Tank_Sta.LB_OFF )
      wire#w2
      R_Coil( #Tank_Sta.Agi_ON )
   END_RUNG
   RUNG wire#w1
      I_Contact( #Lock )
   END_RUNG wire#w2
   // the same network as SCL:
   IF #Tank_Sta.AwysON AND #Tank_Sta.LB_ON AND #Lock THEN #Tank_Sta.Agi_ON := TRUE; END_IF;
   IF #Tank_Sta.AwysON AND (#Tank_Sta.LB_OFF OR NOT #Lock) THEN #Tank_Sta.Agi_ON := FALSE; END_IF;
END_REGION

REGION Network 5: Product Available
   // #HMI.Cmd.%X2 = Product available
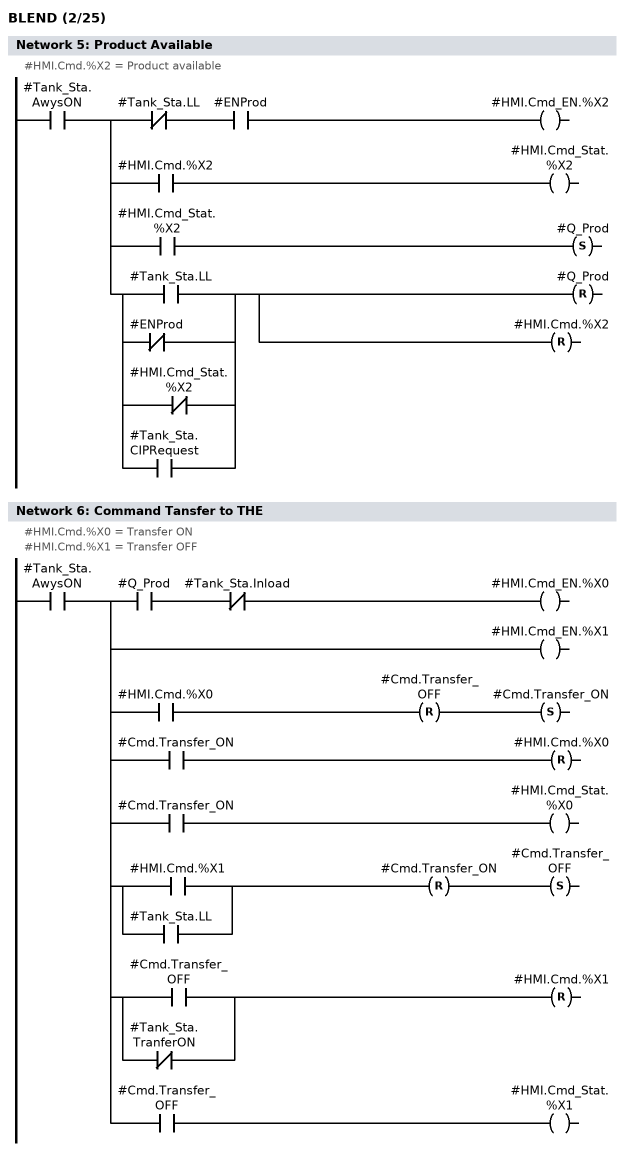
   RUNG wire#powerrail
      Contact( #Tank_Sta.AwysON )
      wire#w1
      I_Contact( #Tank_Sta.LL )
      Contact( #ENProd )
      Coil( #HMI.Cmd_EN.%X2 )
   END_RUNG
   RUNG wire#w1
      Contact( #HMI.Cmd.%X2 )
      Coil( #HMI.Cmd_Stat.%X2 )
   END_RUNG
   RUNG wire#w1
      Contact( #HMI.Cmd_Stat.%X2 )
      S_Coil( #Q_Prod )
   END_RUNG
   RUNG wire#w1
      Contact( #Tank_Sta.LL )
      wire#w2
      R_Coil( #Q_Prod )
   END_RUNG
   RUNG wire#w1
      I_Contact( #ENProd )
   END_RUNG wire#w2
   RUNG wire#w1
      I_Contact( #HMI.Cmd_Stat.%X2 )
   END_RUNG wire#w2
   RUNG wire#w1
      Contact( #Tank_Sta.CIPRequest )
   END_RUNG wire#w2
   RUNG wire#w2
      R_Coil( #HMI.Cmd.%X2 )
   END_RUNG
   // the same network as SCL:
   #HMI.Cmd_EN.%X2 := #Tank_Sta.AwysON AND NOT #Tank_Sta.LL AND #ENProd;
   #HMI.Cmd_Stat.%X2 := #Tank_Sta.AwysON AND #HMI.Cmd.%X2;
   IF #Tank_Sta.AwysON AND #HMI.Cmd_Stat.%X2 THEN #Q_Prod := TRUE; END_IF;
   IF #Tank_Sta.AwysON AND (#Tank_Sta.LL OR NOT #ENProd OR NOT #HMI.Cmd_Stat.%X2 OR #Tank_Sta.CIPRequest) THEN
       #Q_Prod := FALSE;
       #HMI.Cmd.%X2 := FALSE;
   END_IF;
END_REGION

REGION Network 6: Command Tansfer to THE
   // #HMI.Cmd.%X0 = Transfer ON
   // #HMI.Cmd.%X1 = Transfer OFF
   RUNG wire#powerrail
      Contact( #Tank_Sta.AwysON )
      wire#w1
      Contact( #Q_Prod )
      I_Contact( #Tank_Sta.Inload )
      Coil( #HMI.Cmd_EN.%X0 )
   END_RUNG
   RUNG wire#w1
      Coil( #HMI.Cmd_EN.%X1 )
   END_RUNG
   RUNG wire#w1
      Contact( #HMI.Cmd.%X0 )
      R_Coil( #Cmd.Transfer_OFF )
      S_Coil( #Cmd.Transfer_ON )
   END_RUNG
   RUNG wire#w1
      Contact( #Cmd.Transfer_ON )
      R_Coil( #HMI.Cmd.%X0 )
   END_RUNG
   RUNG wire#w1
      Contact( #Cmd.Transfer_ON )
      Coil( #HMI.Cmd_Stat.%X0 )
   END_RUNG
   RUNG wire#w1
      Contact( #HMI.Cmd.%X1 )
      wire#w2
      R_Coil( #Cmd.Transfer_ON )
      S_Coil( #Cmd.Transfer_OFF )
   END_RUNG
   RUNG wire#w1
      Contact( #Tank_Sta.LL )
   END_RUNG wire#w2
   RUNG wire#w1
      Contact( #Cmd.Transfer_OFF )
      wire#w3
      R_Coil( #HMI.Cmd.%X1 )
   END_RUNG
   RUNG wire#w1
      I_Contact( #Tank_Sta.TranferON )
   END_RUNG wire#w3
   RUNG wire#w1
      Contact( #Cmd.Transfer_OFF )
      Coil( #HMI.Cmd_Stat.%X1 )
   END_RUNG
   // the same network as SCL:
   #HMI.Cmd_EN.%X0 := #Tank_Sta.AwysON AND #Q_Prod AND NOT #Tank_Sta.Inload;
   #HMI.Cmd_EN.%X1 := #Tank_Sta.AwysON;
   IF #Tank_Sta.AwysON AND #HMI.Cmd.%X0 THEN
       #Cmd.Transfer_OFF := FALSE;
       #Cmd.Transfer_ON := TRUE;
   END_IF;
   IF #Tank_Sta.AwysON AND #Cmd.Transfer_ON THEN #HMI.Cmd.%X0 := FALSE; END_IF;
   #HMI.Cmd_Stat.%X0 := #Tank_Sta.AwysON AND #Cmd.Transfer_ON;
   IF #Tank_Sta.AwysON AND (#HMI.Cmd.%X1 OR #Tank_Sta.LL) THEN
       #Cmd.Transfer_ON := FALSE;
       #Cmd.Transfer_OFF := TRUE;
   END_IF;
   IF #Tank_Sta.AwysON AND (#Cmd.Transfer_OFF OR NOT #Tank_Sta.TranferON) THEN #HMI.Cmd.%X1 := FALSE; END_IF;
   #HMI.Cmd_Stat.%X1 := #Tank_Sta.AwysON AND #Cmd.Transfer_OFF;
END_REGION

REGION Network 7: Tansfer to THE
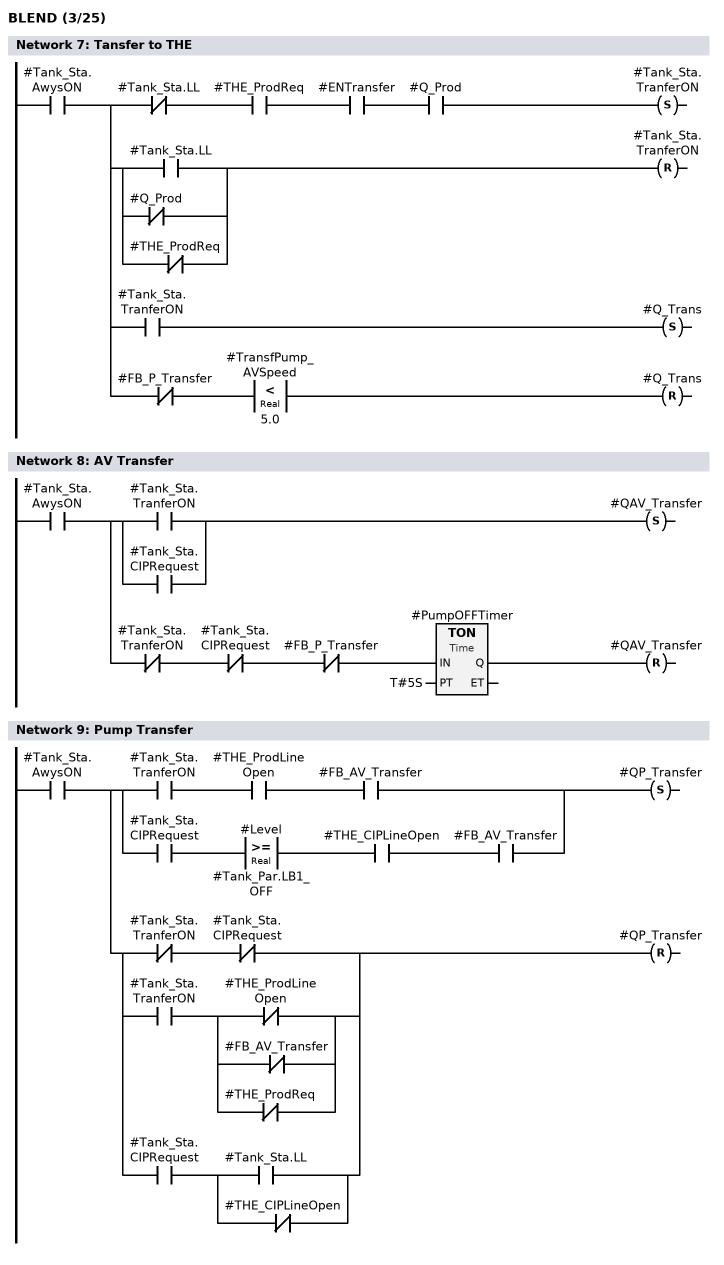
   RUNG wire#powerrail
      Contact( #Tank_Sta.AwysON )
      wire#w1
      I_Contact( #Tank_Sta.LL )
      Contact( #THE_ProdReq )
      Contact( #ENTransfer )
      Contact( #Q_Prod )
      S_Coil( #Tank_Sta.TranferON )
   END_RUNG
   RUNG wire#w1
      Contact( #Tank_Sta.LL )
      wire#w2
      R_Coil( #Tank_Sta.TranferON )
   END_RUNG
   RUNG wire#w1
      I_Contact( #Q_Prod )
   END_RUNG wire#w2
   RUNG wire#w1
      I_Contact( #THE_ProdReq )
   END_RUNG wire#w2
   RUNG wire#w1
      Contact( #Tank_Sta.TranferON )
      S_Coil( #Q_Trans )
   END_RUNG
   RUNG wire#w1
      I_Contact( #FB_P_Transfer )
      { S7_Templates := "SrcType := Real" } LT_Contact(in1 := #TransfPump_AVSpeed, in2 := 5.0)
      R_Coil( #Q_Trans )
   END_RUNG
   // the same network as SCL:
   IF #Tank_Sta.AwysON AND NOT #Tank_Sta.LL AND #THE_ProdReq AND #ENTransfer AND #Q_Prod THEN
       #Tank_Sta.TranferON := TRUE;
   END_IF;
   IF #Tank_Sta.AwysON AND (#Tank_Sta.LL OR NOT #Q_Prod OR NOT #THE_ProdReq) THEN
       #Tank_Sta.TranferON := FALSE;
   END_IF;
   IF #Tank_Sta.AwysON AND #Tank_Sta.TranferON THEN #Q_Trans := TRUE; END_IF;
   IF #Tank_Sta.AwysON AND NOT #FB_P_Transfer AND (#TransfPump_AVSpeed < 5.0) THEN #Q_Trans := FALSE; END_IF;
END_REGION

REGION Network 8: AV Transfer
   RUNG wire#powerrail
      Contact( #Tank_Sta.AwysON )
      wire#w1
      Contact( #Tank_Sta.TranferON )
      wire#w2
      S_Coil( #QAV_Transfer )
   END_RUNG
   RUNG wire#w1
      Contact( #Tank_Sta.CIPRequest )
   END_RUNG wire#w2
   RUNG wire#w1
      I_Contact( #Tank_Sta.TranferON )
      I_Contact( #Tank_Sta.CIPRequest )
      I_Contact( #FB_P_Transfer )
      { S7_Templates := "time_type := Time" } #PumpOFFTimer.TON(pt := T#5S, et =>)
      R_Coil( #QAV_Transfer )
   END_RUNG
   // the same network as SCL:
   IF #Tank_Sta.AwysON AND (#Tank_Sta.TranferON OR #Tank_Sta.CIPRequest) THEN #QAV_Transfer := TRUE; END_IF;
   #PumpOFFTimer(IN := #Tank_Sta.AwysON AND NOT #Tank_Sta.TranferON AND NOT #Tank_Sta.CIPRequest AND NOT #FB_P_Transfer,   // TON
                 PT := T#5S);
   IF #PumpOFFTimer.Q THEN #QAV_Transfer := FALSE; END_IF;
END_REGION

REGION Network 9: Pump Transfer
   RUNG wire#powerrail
      Contact( #Tank_Sta.AwysON )
      wire#w1
      Contact( #Tank_Sta.TranferON )
      Contact( #THE_ProdLineOpen )
      Contact( #FB_AV_Transfer )
      wire#w2
      S_Coil( #QP_Transfer )
   END_RUNG
   RUNG wire#w1
      Contact( #Tank_Sta.CIPRequest )
      { S7_Templates := "SrcType := Real" } GE_Contact(in1 := #Level, in2 := #Tank_Par.LB1_OFF)
      Contact( #THE_CIPLineOpen )
      Contact( #FB_AV_Transfer )
   END_RUNG wire#w2
   RUNG wire#w1
      I_Contact( #Tank_Sta.TranferON )
      I_Contact( #Tank_Sta.CIPRequest )
      wire#w3
      R_Coil( #QP_Transfer )
   END_RUNG
   RUNG wire#w1
      Contact( #Tank_Sta.TranferON )
      wire#w4
      I_Contact( #THE_ProdLineOpen )
   END_RUNG wire#w3
   RUNG wire#w4
      I_Contact( #FB_AV_Transfer )
   END_RUNG wire#w3
   RUNG wire#w4
      I_Contact( #THE_ProdReq )
   END_RUNG wire#w3
   RUNG wire#w1
      Contact( #Tank_Sta.CIPRequest )
      wire#w5
      Contact( #Tank_Sta.LL )
   END_RUNG wire#w3
   RUNG wire#w5
      I_Contact( #THE_CIPLineOpen )
   END_RUNG wire#w3
   // the same network as SCL:
   IF #Tank_Sta.AwysON AND ((#Tank_Sta.TranferON AND #THE_ProdLineOpen AND #FB_AV_Transfer) OR (#Tank_Sta.CIPRequest AND (#Level >= #Tank_Par.LB1_OFF) AND #THE_CIPLineOpen AND #FB_AV_Transfer)) THEN
       #QP_Transfer := TRUE;
   END_IF;
   IF #Tank_Sta.AwysON AND ((NOT #Tank_Sta.TranferON AND NOT #Tank_Sta.CIPRequest) OR (#Tank_Sta.TranferON AND (NOT #THE_ProdLineOpen OR NOT #FB_AV_Transfer OR NOT #THE_ProdReq)) OR (#Tank_Sta.CIPRequest AND (#Tank_Sta.LL OR NOT #THE_CIPLineOpen))) THEN
       #QP_Transfer := FALSE;
   END_IF;
END_REGION

REGION Network 10: CIP Request
   // #HMI.Cmd.%X4 = CIP Request ON
   // #HMI.Cmd.%X5 = CIP Request OFF
